# B&R Automation Studio project Soiled_PLC (part 14)

#### pc.st - Implementation code
```iecst
(********************************************************************
 * COPYRIGHT --
 ********************************************************************
 * Program: pr
 * File: pr.st
 * Author: treamsbottom
 * Created: July 16, 2015
 ********************************************************************
 * Implementation of program pr
 ********************************************************************)
//V1.00.1 First Release
PROGRAM _INIT
//Configuration
mySeq						:= 10;		//Sequence number
myIO						:= 191;
myX20IO						:= 6;		// IO for hardwired stops
myPC						:= 1;
myZone						:= 0;
myRelLine					:= 22;
useRequest					:= FALSE; 	//Use the Request bit. Only use when working with x_1_point. otherwise use RequestRelease as the i_bagAtBuffer.
myBuffBag					:= 0; 		//Buffer bag
myBag						:= 255; 	//Buffer Bag
bufferSettleTime			:= 300;

isDecline					:= FALSE; // VC is moving bags down
myOutBag 					:= Line[myRelLine].LastBag;
END_PROGRAM

PROGRAM _CYCLIC
//Inputs
i_carrAtTop					:= X[myIO].X01;
i_carrAtBottom				:= X[myIO].X02;
i_bagArrive					:= X[myIO].X03;
i_bagOnCarriage				:= X[myIO].X04;
i_bagAtBuffer				:= X[myIO].X05;

i_bagAtBufferOut 		:= FALSE; // Any Single bag buffer out IO.
i_bufferOutOpen			:= FALSE;

o_openBuffer			:= FALSE;
o_openCarriageStop		:= FALSE;
moveToIncomingPosition	:= FALSE;
moveToOutgoingPosition	:= FALSE;

Request.PC[myPC]		:= FALSE;
RequestRel.PC[myPC]		:= FALSE;

IF (myBag = 0) THEN
	Alarm[mySeq].Bag	:= mySeq + 10000;
ELSE
	Alarm[mySeq].Bag	:= myBag;
END_IF;

Alarm[mySeq].Name 		:= 0;
Alarm[mySeq].Beacon		:= TRUE;
Alarm[mySeq].Extra		:= 0;
Alarm[mySeq].Time		:= 3000;

//Setup Sequence
step := D[900 + mySeq];
//Setup Pulse contact
pls := (step <> lastStep);
lastStep := step;

//Sequence
IF (step = 0) THEN
	//Disabled
END_IF;

//Step 1 move to bag in position
IF (step = 1) THEN
	moveToIncomingPosition := TRUE;
	IF carrInIncomingPos THEN
		D[900 + mySeq] := 2;
	END_IF
	IF NOT Std.HaltSysZone[myZone] THEN
		Alarm[mySeq].Name := ALM_CARRIAGE_MOVE_FAULT;
	END_IF;
END_IF;

//Wait for at buffer
ton_10ms_SettledBuffer(IN:= i_bagAtBuffer, PT:= bufferSettleTime);
IF (step = 2) THEN
	moveToIncomingPosition := TRUE;
	IF carrInIncomingPos AND NOT Std.HaltSysZone[myZone] AND NOT i_bagOnCarriage AND NOT i_bagArrive THEN
		IF useRequest THEN
			D[900 + mySeq] := 3;
		ELSE
			IF ton_10ms_SettledBuffer.Q THEN
				IF (myBuffBag > 0) THEN
					IF (Bag[myBuffBag].Cat > 0) AND (Bag[myBag].Cat = 0) THEN
						D[900 + mySeq] := 3;
					ELSIF (Bag[myBuffBag].Cat = 0) THEN
						Alarm[mySeq].Name := ALM_BAG_DATA_ERROR;
						Alarm[mySeq].Bag := myBuffBag;
					ELSE
						Alarm[mySeq].Name := ALM_BAG_DATA_ERROR;
					END_IF;
				ELSE
					D[900 + mySeq] := 3;
				END_IF;
			ELSIF (myBuffBag > 0) AND (Bag[myBuffBag].Cat > 0) THEN
				Alarm[mySeq].Name := ALM_BAG_NOT_SETTLED;
			END_IF;
		END_IF;
	ELSIF NOT Std.HaltSysZone[myZone] THEN
		Alarm[mySeq].Name := ALM_SWITCH_FAULT;
	END_IF;
END_IF;

//Open Buffer stop
IF (step = 3) THEN
	moveToIncomingPosition := TRUE;
	IF carrInIncomingPos THEN
		carrInPosLatch := TRUE;
	END_IF;
	releaseValid := (carrInPosLatch AND ((myBag = 0) OR ((Bag[myBag].Cat = 0) AND (Bag[myBuffBag].Cat > 0))));
	o_openBuffer	   := releaseValid AND NOT useRequest;
	Request.PC[myPC]  := releaseValid AND useRequest;
	IF ((i_bagArrive OR i_bagOnCarriage) AND releaseValid) THEN
		IF (myBag > 0) THEN
			Bag[myBag] := Bag[myBuffBag]; //Clear empty buffer bag data if used
			Bag[myBuffBag] := Bag[0];
		END_IF;
		D[900 + mySeq] := 4;
	ELSIF (myBag > 0) THEN
		IF (Bag[myBag].Cat > 0) THEN
			Alarm[mySeq].Name := ALM_BAG_DATA_ERROR;
			Alarm[mySeq].Time := 0;
		ELSIF (Bag[myBuffBag].Cat = 0) THEN
			Alarm[mySeq].Name := ALM_BAG_DATA_ERROR;
			Alarm[mySeq].Bag := myBuffBag;
			Alarm[mySeq].Time := 0;
		ELSE
			Alarm[mySeq].Name  := ALM_BAG_NOT_ARRIVED;
		END_IF;
	ELSIF NOT carrInPosLatch THEN
		Alarm[mySeq].Name  := ALM_SWITCH_FAULT;
	ELSE
		Alarm[mySeq].Name  := ALM_BAG_NOT_ARRIVED;
	END_IF;
END_IF;

// Step 4 Bag settles on carriage..
ton_10ms_SettledCarriage(IN:= i_bagOnCarriage, PT:= 300);
IF (step = 4) THEN
	moveToIncomingPosition := TRUE;
	IF  ton_10ms_SettledCarriage.Q AND NOT Std.HaltSysZone[myZone] AND NOT i_bagArrive THEN
		D[900 + mySeq] := 5;
	ELSIF NOT Std.HaltSysZone[myZone] THEN
		Alarm[mySeq].Name := ALM_BAG_NOT_SETTLED;
	END_IF;
END_IF

// Step 5 move to outgoing position
IF (step = 5) THEN
	moveToOutgoingPosition := TRUE;
	IF carrAtOutgoingPos THEN
		D[900 + mySeq] := 6;
	ELSIF NOT Std.HaltSysZone[myZone] THEN
		Alarm[mySeq].Name := ALM_CARRIAGE_MOVE_FAULT;
	END_IF;
END_IF;

//Step 6 check release condtion.
//Check for line space.
IF (step = 6) THEN
	moveToOutgoingPosition := TRUE;
	releaseValid := (carrAtOutgoingPos AND NOT i_bagAtBufferOut AND NOT i_bufferOutOpen AND ((myBag = 0) OR ((Bag[myBag].Cat > 0) AND (Bag[myOutBag].Cat = 0))));
	IF (myRelLine > 0) THEN
		IF (Line[myRelLine].Clear AND releaseValid) THEN
			C[myRelLine] := 0;
			D[900 + mySeq] := 7;
		END_IF;
		IF NOT carrAtOutgoingPos THEN
			Alarm[mySeq].Name := ALM_CARRIAGE_MOVE_FAULT;
			Alarm[mySeq].Time := 0;
		ELSIF (Line[myRelLine].Clear AND i_bagAtBufferOut) THEN
			Alarm[mySeq].Name := ALM_SWITCH_FAULT;
		ELSIF (myBag > 0) AND (Bag[myBag].Cat = 0) THEN
			Alarm[mySeq].Name := ALM_BAG_DATA_ERROR;
			Alarm[mySeq].Time := 0;
		ELSIF Line[myRelLine].Clear AND (myOutBag > 0) AND (Bag[myOutBag].Cat > 0) THEN
			Alarm[mySeq].Name := ALM_BAG_DATA_ERROR;
			Alarm[mySeq].Bag := myOutBag;
			Alarm[mySeq].Time := 0;
		END_IF;
	ELSE
		RequestRel.PC[myPC] := releaseValid;
		IF EnableRel.PC[myPC] AND releaseValid THEN
			D[900 + mySeq] := 7;
		ELSIF NOT carrAtOutgoingPos THEN
			Alarm[mySeq].Name := ALM_CARRIAGE_MOVE_FAULT;
			Alarm[mySeq].Time := 0;
		ELSIF (myBag > 0) AND (Bag[myBag].Cat = 0) THEN
			Alarm[mySeq].Name := ALM_BAG_DATA_ERROR;
			Alarm[mySeq].Time := 0;
		ELSIF (myOutBag > 0) AND (Bag[myOutBag].Cat > 0) THEN
			Alarm[mySeq].Name := ALM_BAG_DATA_ERROR;
			Alarm[mySeq].Bag := myOutBag;
			Alarm[mySeq].Time := 0;
		END_IF;
	END_IF;
END_IF;

//Step 7 Release bag.
IF (step = 7) THEN
	releaseValid := (NOT i_bagAtBufferOut AND NOT i_bufferOutOpen AND ((myBag = 0) OR ((Bag[myBag].Cat > 0) AND (Bag[myOutBag].Cat = 0))));
	o_openCarriageStop := releaseValid AND NOT Std.HaltSysZone[myZone];
	IF releaseValid THEN
		IF (myBag = 0) THEN
			IF (myRelLine > 0) THEN
				IF Line[myRelLine].Trip THEN
					D[900 + mySeq] := 1;
				END_IF;
			ELSE
				IF NOT EnableRel.PC[myPC] THEN
					D[900 + mySeq] := 1;
				END_IF;
			END_IF;
			IF NOT Std.HaltSysZone[myZone] THEN
				Alarm[mySeq].Name := ALM_BAG_NOT_RELEASED;
			END_IF;
		ELSE//Use tracking
			IF (myRelLine > 0) THEN
				IF Line[myRelLine].Trip THEN
					Bag[myOutBag] := Bag[myBag];
					Bag[myBag] := Bag[0];
					D[900 + mySeq] := 1;
				END_IF;
			ELSE
				IF NOT EnableRel.PC[myPC] AND (Bag[myBag].Cat = 0) THEN // Make sure data is copied out by enabling sequence.
					D[900 + mySeq] := 1;
				ELSIF NOT EnableRel.PC[myPC] AND (Bag[myBag].Cat > 0) THEN
					Alarm[mySeq].Name := ALM_BAG_DATA_ERROR;
				END_IF;
			END_IF;
		END_IF;
	ELSIF NOT carrAtOutgoingPos THEN
		Alarm[mySeq].Name := ALM_CARRIAGE_MOVE_FAULT;
		Alarm[mySeq].Time := 0;
	ELSIF i_bagAtBufferOut AND NOT i_bufferOutOpen THEN
		Alarm[mySeq].Name := ALM_SWITCH_FAULT;
		Alarm[mySeq].Time := 0;
	ELSIF (myBag > 0) THEN
		IF (Bag[myBag].Cat = 0) THEN
			Alarm[mySeq].Name := ALM_BAG_DATA_ERROR;
			Alarm[mySeq].Time := 0;
		ELSIF (Bag[myOutBag].Cat > 0) THEN
			Alarm[mySeq].Name := ALM_BAG_DATA_ERROR;
			Alarm[mySeq].Bag := myOutBag;
			Alarm[mySeq].Time := 0;
		END_IF;
	END_IF;
END_IF;

//Control Position
IF isDecline THEN
	o_moveUp := moveToIncomingPosition;
	o_moveDown := moveToOutgoingPosition;
	carrInIncomingPos := i_carrAtTop;
	carrAtOutgoingPos := i_carrAtBottom;
ELSE
	o_moveDown := moveToIncomingPosition;
	o_moveUp := moveToOutgoingPosition;
	carrInIncomingPos := i_carrAtBottom;
	carrAtOutgoingPos := i_carrAtTop;
END_IF;

//-----------------------------------
//PLC Outputs - adjust TO suit system
//-----------------------------------

Y[myIO].Y06			:= o_openBuffer;
Y[myIO].Y07			:= ((step >= 3) AND (step <= 4) AND carrInIncomingPos); //Safe stop

Y[myX20IO].Y01 		:= (o_moveUp AND NOT i_carrAtTop); //Move carriage up
Y[myX20IO].Y02 		:= (o_moveDown  AND NOT i_carrAtBottom);//Move carriage down
Y[myX20IO].Y03 		:= (o_openCarriageStop AND carrAtOutgoingPos);// Carriage Stop

//Don't allow forcing of carriage movement and carriage stop
YForceDisable[myX20IO].Y01 	:= TRUE;
YForceDisable[myX20IO].Y02 	:= TRUE;
YForceDisable[myX20IO].Y03 	:= TRUE;

//Alarms
timerAlarm(IN := NOT pls AND (Alarm[mySeq].Name > 0),PT:= Alarm[mySeq].Time);

Alarm[mySeq].On 	:= timerAlarm.Q;
Alarm[mySeq].ET 	:= timerAlarm.ET;

END_PROGRAM
```

### Program Logical/BaseStandards/Pneumatic/pic (IEC, version 1.00.3) - *Pneumatic Incline

#### pic.st - Implementation code
```iecst
(********************************************************************
 * COPYRIGHT --
 ********************************************************************
 * Program: pic
 * File: pic.st
 * Author: treamsbottom
 * Created: July 16, 2015
 ********************************************************************
 * Implementation of program pic - Pneumatic Incline
 ********************************************************************)
//V1.00.1 First Release
PROGRAM _INIT
//Configuration
mySeq						:= 22;	//Sequence number
myIO						:= 201;
myZone						:= 0;
myRelLine					:= 22;
myBuffBag					:= 0;
myBag						:= 0;
bufferSettleTime			:= 300;
myPI						:= 1;

myOutBag 					:= Line[myRelLine].LastBag;
END_PROGRAM

PROGRAM _CYCLIC
//Inputs

i_bagInIncline			:= X[myIO].X01;
i_cylinderAtBottom		:= X[myIO].X02;
i_cylinderAtTop			:= X[myIO].X03;
i_bagAtBuffer			:= X[myIO].X04;

i_bagAtBufferOut 		:= FALSE; // Any Single bag buffer out IO.
i_bufferOutOpen			:= FALSE;

o_openBuffer			:= FALSE;
o_cylinderDown			:= FALSE;

Request.PI[myPI]		:= FALSE;
RequestRel.PI[myPI]		:= FALSE;

IF (myBag = 0) THEN
	Alarm[mySeq].Bag	:= mySeq + 10000;
ELSE
	Alarm[mySeq].Bag	:= myBag;
END_IF;

Alarm[mySeq].Name 		:= 0;
Alarm[mySeq].Beacon	:= TRUE;
Alarm[mySeq].Extra		:= 0;
Alarm[mySeq].Time		:= 3000;

//Setup Sequence
step := D[900 + mySeq];
//Setup Pulse contact
pls := (step <> lastStep);
lastStep := step;

//Sequence
IF (step = 0) THEN
	//Disabled
END_IF;

//Wait for at buffer
ton_10ms_SettledBuffer(IN:= i_bagAtBuffer, PT:= bufferSettleTime);
IF (step = 1) THEN
	IF NOT Std.HaltSysZone[myZone] AND i_cylinderAtTop AND NOT i_bagInIncline THEN
		IF useRequest THEN
			D[900 + mySeq] := 2;
		ELSE
			IF ton_10ms_SettledBuffer.Q THEN
				IF (myBuffBag > 0) THEN
					IF (Bag[myBuffBag].Cat > 0) AND (Bag[myBag].Cat = 0) THEN
						D[900 + mySeq] := 2;
					ELSIF (Bag[myBuffBag].Cat = 0) THEN
						Alarm[mySeq].Name := ALM_BAG_DATA_ERROR;
						Alarm[mySeq].Bag := myBuffBag;
					ELSE
						Alarm[mySeq].Name := ALM_BAG_DATA_ERROR;
					END_IF;
				ELSE
					D[900 + mySeq] := 2;
				END_IF;
			ELSIF (myBuffBag > 0) AND (Bag[myBuffBag].Cat > 0) THEN
				Alarm[mySeq].Name := ALM_BAG_NOT_SETTLED;
			END_IF;
		END_IF;
	ELSIF NOT Std.HaltSysZone[myZone] THEN
		Alarm[mySeq].Name := ALM_SWITCH_FAULT;
	END_IF;
END_IF;

//Open Buffer stop
IF (step = 2) THEN
	releaseValid := ((myBag = 0) OR ((Bag[myBag].Cat = 0) AND (Bag[myBuffBag].Cat > 0)));
	o_openBuffer	   := releaseValid AND NOT useRequest;
	Request.PI[myPI]  := releaseValid AND useRequest;
	IF (i_bagInIncline AND releaseValid) THEN
		IF (myBag > 0) THEN
			Bag[myBag] := Bag[myBuffBag]; //Clear empty buffer bag data if used
			Bag[myBuffBag] := Bag[0];
		END_IF;
		D[900 + mySeq] := 3;
	ELSIF (myBag > 0) THEN
		IF (Bag[myBag].Cat > 0) THEN
			Alarm[mySeq].Name := ALM_BAG_DATA_ERROR;
			Alarm[mySeq].Time := 0;
		ELSIF (Bag[myBuffBag].Cat = 0) THEN
			Alarm[mySeq].Name := ALM_BAG_DATA_ERROR;
			Alarm[mySeq].Bag := myBuffBag;
			Alarm[mySeq].Time := 0;
		ELSE
			Alarm[mySeq].Name  := ALM_BAG_NOT_ARRIVED;
		END_IF;
		Alarm[mySeq].Name  := ALM_BAG_NOT_ARRIVED;
	END_IF;
END_IF;

//Let bag settle at base OF incline
ton_10ms_SettledInIncline(IN:= i_bagInIncline, PT:= 300);
IF (step = 3) THEN
	o_openBuffer := NOT useRequest;
	IF  ton_10ms_SettledInIncline.Q AND NOT Std.HaltSysZone[myZone] THEN
		D[900 + mySeq] := 4;
	ELSIF NOT Std.HaltSysZone[myZone] THEN
		Alarm[mySeq].Name := ALM_BAG_NOT_SETTLED;
	END_IF;
END_IF

//Move incline down to collect first trolley
ton_10ms_CylinderDown(IN := i_cylinderAtBottom, PT:=300);
IF (step = 4) THEN
	o_openBuffer := NOT useRequest;
	o_cylinderDown := TRUE;
	IF ton_10ms_CylinderDown.Q THEN
		D[900 + mySeq] := 5;
	END_IF;
	Alarm[mySeq].Name := ALM_SWITCH_FAULT;
END_IF;

//Let cylinder move back to the top.
IF (step = 5) THEN
	o_openBuffer := NOT useRequest;
	IF i_cylinderAtTop THEN
		D[900 + mySeq] := 6;
	END_IF;
	Alarm[mySeq].Name := ALM_SWITCH_FAULT;
END_IF;

//Check for valid release..
//Check for line space.
IF (step = 6) THEN
	releaseValid := (ton_10ms_SettledInIncline.Q AND NOT i_cylinderAtBottom AND NOT i_bagAtBufferOut AND NOT i_bufferOutOpen AND ((myBag = 0) OR ((Bag[myBag].Cat > 0) AND (Bag[myOutBag].Cat = 0))));
	IF (myRelLine > 0) THEN
		IF (Line[myRelLine].Clear AND releaseValid) THEN
			C[myRelLine] := 0;
			D[900 + mySeq] := 7;
		END_IF;
		IF i_cylinderAtBottom OR NOT i_bagInIncline THEN
			Alarm[mySeq].Name := ALM_SWITCH_FAULT;
			Alarm[mySeq].Time := 0;
		ELSIF (Line[myRelLine].Clear AND i_bagAtBufferOut) THEN
			Alarm[mySeq].Name := ALM_SWITCH_FAULT;
		ELSIF (myBag > 0) AND (Bag[myBag].Cat = 0) THEN
			Alarm[mySeq].Name := ALM_BAG_DATA_ERROR;
			Alarm[mySeq].Time := 0;
		ELSIF Line[myRelLine].Clear AND (myOutBag > 0) AND (Bag[myOutBag].Cat > 0) THEN
			Alarm[mySeq].Name := ALM_BAG_DATA_ERROR;
			Alarm[mySeq].Bag := myOutBag;
			Alarm[mySeq].Time := 0;
		END_IF;
	ELSE
		RequestRel.PI[myPI] := releaseValid;
		IF EnableRel.PI[myPI] AND releaseValid THEN
			D[900 + mySeq] := 7;
		ELSIF NOT i_cylinderAtBottom OR NOT i_bagInIncline THEN
			Alarm[mySeq].Name := ALM_SWITCH_FAULT;
			Alarm[mySeq].Time := 0;
		ELSIF (myBag > 0) AND (Bag[myBag].Cat = 0) THEN
			Alarm[mySeq].Name := ALM_BAG_DATA_ERROR;
			Alarm[mySeq].Time := 0;
		ELSIF (myOutBag > 0) AND (Bag[myOutBag].Cat > 0) THEN
			Alarm[mySeq].Name := ALM_BAG_DATA_ERROR;
			Alarm[mySeq].Bag := myOutBag;
			Alarm[mySeq].Time := 0;
		END_IF;
	END_IF;
END_IF;

//Move cylinder down to get 2nd trolley.
IF (step = 7) THEN
	o_cylinderDown := TRUE;
	IF  ton_10ms_CylinderDown.Q THEN
		D[900 + mySeq] := 8;
	END_IF;
	Alarm[mySeq].Name := ALM_SWITCH_FAULT;
END_IF;

//Release bag
IF (step = 8) THEN
	releaseValid := (NOT i_bagAtBufferOut AND NOT i_bufferOutOpen AND ((myBag = 0) OR ((Bag[myBag].Cat > 0) AND (Bag[myOutBag].Cat = 0))));
	o_cylinderDown := NOT releaseValid; // Hold cylinder down if release is not valid.
	IF releaseValid THEN
		IF (myBag = 0) THEN// Not tracking.
			IF (myRelLine > 0) THEN
				IF Line[myRelLine].Trip THEN
					D[900 + mySeq] := 1;
				END_IF;
			ELSE
				IF NOT EnableRel.PI[myPI] THEN
					D[900 + mySeq] := 1;
				END_IF;
			END_IF;
			IF NOT Std.HaltSysZone[myZone] THEN
				Alarm[mySeq].Name := ALM_BAG_NOT_RELEASED;
			END_IF;
		ELSE//Use tracking
			IF (myRelLine > 0) THEN
				IF Line[myRelLine].Trip THEN
					Bag[myOutBag] := Bag[myBag];
					Bag[myBag] := Bag[0];
					D[900 + mySeq] := 1;
				END_IF;
			ELSE
				IF NOT EnableRel.PI[myPI] AND (Bag[myBag].Cat = 0) THEN // Make sure data is copied out by enabling sequence.
					D[900 + mySeq] := 1;
				ELSIF NOT EnableRel.PI[myPI] AND (Bag[myBag].Cat > 0) THEN
					Alarm[mySeq].Name := ALM_BAG_DATA_ERROR;
				END_IF;
			END_IF;
		END_IF;
	ELSIF i_bagAtBufferOut AND NOT i_bufferOutOpen THEN
		Alarm[mySeq].Name := ALM_SWITCH_FAULT;
		Alarm[mySeq].Time := 0;
	ELSIF (myBag > 0) THEN
		IF (Bag[myBag].Cat = 0) THEN
			Alarm[mySeq].Name := ALM_BAG_DATA_ERROR;
			Alarm[mySeq].Time := 0;
		ELSIF (Bag[myOutBag].Cat > 0) THEN
			Alarm[mySeq].Name := ALM_BAG_DATA_ERROR;
			Alarm[mySeq].Bag := myOutBag;
			Alarm[mySeq].Time := 0;
		END_IF;
	END_IF;
END_IF

//-----------------------------------
//PLC Outputs - adjust TO suit system
//-----------------------------------

Y[myIO].Y05 := o_cylinderDown;
Y[myIO].Y06 := o_openBuffer;

//Alarms
timerAlarm(IN := NOT pls AND (Alarm[mySeq].Name > 0),PT:= Alarm[mySeq].Time);

Alarm[mySeq].On 	:= timerAlarm.Q;
Alarm[mySeq].ET 	:= timerAlarm.ET;

END_PROGRAM
```

### Package Logical/BaseStandards/Misc - Misc - Speed Reducer,Pressure relief

### Program Logical/BaseStandards/Misc/ssr (IEC, version 1.00.1) - speed reducer

- Standard Sequence Speed Reducer V1.00.1 ENG.docx (binary file, 203679 bytes)
#### ssr.st - Implementation code
```iecst
(********************************************************************
 * COPYRIGHT --
 ********************************************************************
 * Program: ssr
 * File: ssr.st
 * Author: treamsbottom
 * Created: July 16, 2015
 ********************************************************************
 * Implementation of program ssr
 ********************************************************************)
//V1.00.1 FIRST VERSION
PROGRAM _INIT

END_PROGRAM

PROGRAM _CYCLIC

myHaltSys				:= Std.HaltSysZone[0];

//Inputs
i_bagApproach[1]		:= X[212].X01;

FOR n := 1 TO LOCAL_MAX_SPEED_REDUCERS DO

	ctu_tripCount[n](CU	:= i_bagApproach[n],PV := 2,RESET := ton_10ms_openBrush[n].Q);
	ton_10ms_openBrush[n](IN := NOT myHaltSys AND o_closeBrush[n],PT	:= 300);

	IF (ctu_tripCount[n].CV >= 2) THEN
		o_closeBrush[n] := TRUE;
	END_IF;

	IF ton_10ms_openBrush[n].Q THEN
		o_closeBrush[n] := FALSE;
	END_IF;
END_FOR;

//Outputs
Y[212].Y05		:= o_closeBrush[1];

END_PROGRAM
```

#### ssr.var - Local variables
```iecst
(********************************************************************
 * COPYRIGHT --
 ********************************************************************
 * Program: ssr
 * File: ssr.var
 * Author: treamsbottom
 * Created: July 16, 2015
 ********************************************************************
 * Local variables of program ssr
 ********************************************************************)
VAR
	myHaltSys : BOOL;
	i_bagApproach : ARRAY[0..LOCAL_MAX_SPEED_REDUCERS] OF BOOL;
	n : UINT;
	ctu_tripCount : ARRAY[0..LOCAL_MAX_SPEED_REDUCERS] OF CTU;
	ton_10ms_openBrush : ARRAY[0..LOCAL_MAX_SPEED_REDUCERS] OF TON_10ms;
	o_closeBrush : ARRAY[0..LOCAL_MAX_SPEED_REDUCERS] OF BOOL;
END_VAR
VAR CONSTANT
	LOCAL_MAX_SPEED_REDUCERS : UINT := 1;
END_VAR
```

### Package Logical/BaseStandards/Sorting - *All sorting equipment

### Program Logical/BaseStandards/Sorting/zzCustomerChange (IEC)

#### zzCustomerChange.ab - Implementation code
```automation-basic
(********************************************************************
 * COPYRIGHT -- HP
 ********************************************************************
 * Program: zzCustomerChange
 * File: zzCustomerChange.ab
 * Author: treamsbottom
 * Created: November 18, 2014
 ********************************************************************
 * Implementation of program zzCustomerChange
 ********************************************************************)

PROGRAM _INIT

END_PROGRAM

 PROGRAM _CYCLIC
; Multiple Bank Customer change,UINT
; Use D32[80 + Bank] to send new customer
; Use D32[90 + Bank] for reply

myZone 			= 0
mySeq			= 83
;I_PxStart_Belt[3] = X[3].X04;belt blocked
I_PxEnd_Belt[3] = NOT X[350].X01
I_PxEnd_Belt[4] = NOT X[351].X01
I_PxEnd_Belt[5] = NOT X[351].X02
I_PxEnd_Belt[7] = NOT X[350].X03
I_PxEnd_Belt[8] = NOT X[351].X03
I_PxEnd_Belt[9] = NOT X[351].X04
I_PxEnd_Belt[11] = NOT X[350].X04
I_PxEnd_Belt[12] = NOT X[350].X02

I_InvStatus[2]	= X[360].X06 OR DebugMode
I_InvStatus[3]	= X[360].X07 OR DebugMode
I_InvStatus[4]	= X[360].X08 OR DebugMode
I_InvStatus[5]	= X[361].X01 OR DebugMode
I_InvStatus[7]	= X[361].X02 OR DebugMode
I_InvStatus[8]	= X[361].X03 OR DebugMode
I_InvStatus[9]	= X[361].X04 OR DebugMode
I_InvStatus[11]	= X[361].X05 OR DebugMode
I_InvStatus[12]	= X[361].X06 OR DebugMode

I_MultipleCustomers = (D[900 +  mySeq] = 1)

I_AcceptNewCustomer[1] = X[3].X07
I_AcceptNewCustomer[2] = X[3].X08

myCustBag[1] = 471
myNewCustBag[1] = 472
myCustBag[2] = 473
myNewCustBag[2] = 474

Alarm[mySeq].Name 				= 0
Alarm[mySeq].Bag				= 10083
Alarm[mySeq].Beacon				= TRUE
Alarm[mySeq].Extra				= 0
Alarm[mySeq].Time			  	= 500

LOOP n = 1 TO MAX_BANKS DO
	Bag[myCustBag[n]].Prg = 1
	Bag[myCustBag[n]].Cat = 1 ; Force Cat to stop bag being deleted
	Bag[myCustBag[n]].Bid = n
	Bag[myNewCustBag[n]].Prg = 1
	Bag[myNewCustBag[n]].Cat = 1
	Bag[myNewCustBag[n]].Bid = n+10
	O_CustChange_Lamp[n] = FALSE
	O_CustChange_Piezo[n] = FALSE
	RunBelts[n]	= FALSE
ENDLOOP

LOOP n = 1 TO MAX_BELTS DO
	O_RunBelt[n] = FALSE
	O_SlowBelt[n] = FALSE
ENDLOOP

O_Extend[1] = FALSE
O_Extend[2] = FALSE

O_Retract[1] = FALSE
O_Retract[2] = FALSE

SortingEnable = (D[3] > 0) AND NOT Std.HaltSysZone[myZone]

	;Local Vars for each bank End of first set of sorting belts..
I_End_1st_Belt[1] 		= I_PxEnd_Belt[3]
I_End_1st_Belt[2] 		= I_PxEnd_Belt[7]
;LOOP t = 1 TO 6 DO
;	TON_BeltBlocked[t].IN = I_PxStart_Belt[t]
;	TON_BeltBlocked[t].PT = 150
;	TON_BeltBlocked[t] FUB TON_10ms()
;ENDLOOP
;LOOP t = 1 TO MAX_BANKS DO; IF both px are made and belt is running for more than 6 secs then pulse belt
;
;	TON_RestartBelts[t].IN = (O_RunBelt[t * 3] AND NOT TON_BeltBlocked[t * 3].Q)
;	TON_RestartBelts[t].PT = 300
;	TON_RestartBelts[t] FUB TON_10ms()
;
;	TON_PulseBelt[t].IN = (O_RunBelt[t * 3] AND I_End_1st_Belt[t] AND TON_BeltBlocked[t * 3].Q)
;	TON_PulseBelt[t].PT = 600
;	TON_PulseBelt[t] FUB TON_10ms()
;ENDLOOP
;TON_10ms(NOT PulseOff,500,PulseOn,PulseOnET)
;TON_10ms(PulseOn,200,PulseOff,PulseOffET)

;
;myNextBeltRunning[1]	= ((SortingEnable AND NOT I_End_1st_Belt[1]) OR TON_RestartBelts[1].Q OR (TON_PulseBelt[1].Q AND PulseOn))
;myNextBeltRunning[2]	= ((SortingEnable AND NOT I_End_1st_Belt[2]) OR TON_RestartBelts[2].Q OR (TON_PulseBelt[2].Q AND PulseOn))
;

IF NOT I_MultipleCustomers THEN
	Bag[myNewCustBag[2]].Cus =  Bag[myNewCustBag[1]].Cus
	;CustomerChangeDisplay[2].InputLock = 1	 ;**Is overwritten at end of cyclic code.
ENDIF

LOOP n = 1 TO MAX_BANKS DO
	;Default Display Values
	strcpy(ADR(CustomerChangeDisplay[n].Message),ADR(""))
	CustomerChangeDisplay[n].MessageText_Colour = BgLtGrey + FgBlack
	CustomerChangeDisplay[n].InputLock = 0
	CustomerChangeDisplay[n].InputText_Colour = BgWhite + FgBlack
	CustomerChangeDisplay[n].New_CustomerNo = Bag[myNewCustBag[n]].Cus

	TON_PiezoDelay[n].IN = (CustomerChange[n] = 1)
	TON_PiezoDelay[n].PT = 300
	TON_PiezoDelay[n] FUB TON_10ms()

	IF ((Bag[myNewCustBag[n]].Cus = 0) OR (Bag[myCustBag[n]].Cus = Bag[myNewCustBag[n]].Cus)) THEN
 		CustomerChange[n] = 0
	ENDIF

	CASE CustomerChange[n] OF
		ACTION 0: ; Normal Run Belts as normal
;			strcpy(ADR(CustomerChangeDisplay[n].Message),ADR(""))
;			CustomerChangeDisplay[n].MessageText_Colour = BgLtGrey + FgBlack
;			CustomerChangeDisplay[n].InputLock = 0
;			CustomerChangeDisplay[n].InputText_Colour = BgWhite + FgBlack
			D32[80 + n] = 0
			D32[90 + n] = 0
			RunBelts[n] = SortingEnable
        	IF ((Bag[myCustBag[n]].Cus <> Bag[myNewCustBag[n]].Cus) AND (Bag[myNewCustBag[n]].Cus > 0)) THEN
				CustomerChange[n] = 1
			ENDIF
		ENDACTION

		ACTION 1: ; Stop belt at photocell	and wait for customer change accept.
;			strcpy(ADR(CustomerChangeDisplay[n].Message),ADR("Wait for accept pushbutton"))
;			CustomerChangeDisplay[n].MessageText_Colour = BgLtGrey + FgBlack
;			CustomerChangeDisplay[n].InputLock = 2

			RunBelts[n] = SortingEnable	AND NOT I_End_1st_Belt[n]
			O_CustChange_Lamp[n] = Std.Clock1s
			O_CustChange_Piezo[n] = NOT TON_PiezoDelay[n].Q
			IF I_AcceptNewCustomer[n] THEN
				CustomerChange[n] = 2
			ENDIF
		ENDACTION

		ACTION 2: ;Send new customer request to trackview
			RunBelts[n] = SortingEnable//myNextBeltRunning[n]
			//CustomerChangeDisplay[n].InputLock = 2
			D32[80 + n] = Bag[myNewCustBag[n]].Cus ; Send new customer to trackview

			AutoChangeState = D32[90 + n]
			CASE AutoChangeState OF
				ACTION 0: ;Busy
					//CustomerChangeDisplay[n].MessageText_Colour = BgLtGrey + FgBlack
					//strcpy(ADR(CustomerChangeDisplay[n].Message),ADR("Loading Program - Please Wait"))
					O_CustChange_Lamp[n] = TRUE
					myCustChangeMessageStatus[n] = 99
				ENDACTION

				ACTION 1: ; Ok
					//CustomerChangeDisplay[n].MessageText_Colour = BgLtGrey + FgBlack
					//strcpy(ADR(CustomerChangeDisplay[n].Message),ADR("Program Loaded"))
					Bag[myCustBag[n]].Cus = Bag[myNewCustBag[n]].Cus
					CustomerChange[n] = 0
				ENDACTION

				ACTION 2..3: ; 2 = no program, 3 = invalid
;					IF (AutoChangeState = 2) THEN
;						strcpy(ADR(CustomerChangeDisplay[n].Message),ADR("No Program! Press accept pushbutton"))
;					ELSE
;						strcpy(ADR(CustomerChangeDisplay[n].Message),ADR("Invalid Program! Press accept pushbutton"))
;					ENDIF
;					CustomerChangeDisplay[n].MessageText_Colour = BgLtGrey + FgRed
					O_CustChange_Lamp[n] = Std.Clock500ms
//					myCustChangeMessageStatus[n] = UINT(AutoChangeState)
					IF I_AcceptNewCustomer[n] THEN
						Bag[myCustBag[n]].Cus = Bag[myNewCustBag[n]].Cus
						CustomerChange[n] = 0
					ENDIF
				ENDACTION

				ELSEACTION: ; ERROR!!
				//	strcpy(ADR(CustomerChangeDisplay[n].Message),ADR("ERROR! Press accept pushbutton"))
				//	CustomerChangeDisplay[n].MessageText_Colour = BgLtGrey + FgRed
					O_CustChange_Lamp[n] = Std.Clock500ms
				//	myCustChangeMessageStatus[n] = 4
					IF I_AcceptNewCustomer[n] THEN
						Bag[myCustBag[n]].Cus = Bag[myNewCustBag[n]].Cus
						CustomerChange[n] = 0
					ENDIF
				ENDACTION
			ENDCASE
		ENDACTION

	ENDCASE
ENDLOOP

//**************Belt controls...
	CASE D[983] OF
		ACTION 0://Carousel mode.
			O_Extend[1] = TRUE
			O_Extend[2] = TRUE
        	LOOP n = 1 TO MAX_BELTS DO
				O_RunBelt[n] = SortingEnable AND I_InvStatus[n]
			ENDLOOP
		ENDACTION
		ACTION 1://Retract Both belts
			O_Retract[1] = TRUE
			O_Retract[2] = TRUE
			O_RunBelt[5] =  (SortingEnable AND I_InvStatus[5] AND NOT Stn[41].SP3 AND NOT Stn[41].CloseFlap AND ((Stn[41].QTime = 0) OR NOT I_PxEnd_Belt[5]))
			O_SlowBelt[5] = Stn[41].SP1 AND I_PxEnd_Belt[5]
			O_RunBelt[4] = SortingEnable AND I_InvStatus[4] AND (O_RunBelt[5] OR NOT I_PxEnd_Belt[4])

			O_RunBelt[12] =  (SortingEnable AND I_InvStatus[12] AND NOT Stn[42].SP3 AND NOT Stn[42].CloseFlap AND ((Stn[42].QTime = 0) OR NOT I_PxEnd_Belt[12]))
			O_SlowBelt[12] = Stn[42].SP1 AND I_PxEnd_Belt[12]
			O_RunBelt[11] = SortingEnable AND I_InvStatus[11] AND (O_RunBelt[12] OR NOT I_PxEnd_Belt[11])
			O_RunBelt[9] = SortingEnable AND I_InvStatus[9] AND (O_RunBelt[11] OR NOT I_PxEnd_Belt[9])
			O_RunBelt[8] = SortingEnable AND I_InvStatus[8] AND (O_RunBelt[9] OR NOT I_PxEnd_Belt[8])
		ENDACTION

		ACTION 2://Retract Only SB12
			O_Extend[1] = TRUE
			O_Retract[2] = TRUE
			O_RunBelt[12] =  (SortingEnable AND I_InvStatus[12] AND NOT Stn[42].SP3 AND NOT Stn[42].CloseFlap AND ((Stn[42].QTime = 0) OR NOT I_PxEnd_Belt[12]))
			O_RunBelt[11] = SortingEnable AND I_InvStatus[11] AND (O_RunBelt[12] OR NOT I_PxEnd_Belt[11])
			O_RunBelt[9] = SortingEnable AND I_InvStatus[9] AND (O_RunBelt[11] OR NOT I_PxEnd_Belt[9])
			O_RunBelt[8] = SortingEnable AND I_InvStatus[8] AND (O_RunBelt[9] OR NOT I_PxEnd_Belt[8])

			O_RunBelt[5] = SortingEnable AND I_InvStatus[5] AND (O_RunBelt[10] OR NOT I_PxEnd_Belt[5])
			O_RunBelt[4] = SortingEnable AND I_InvStatus[4] AND (O_RunBelt[5] OR NOT I_PxEnd_Belt[4])
		ENDACTION

		ACTION 3://Retract Only SB5
			O_Retract[1] = TRUE
			O_Extend[2] = TRUE

			O_RunBelt[5] =  (SortingEnable AND I_InvStatus[5] AND NOT Stn[41].SP3 AND NOT Stn[41].CloseFlap AND ((Stn[41].QTime = 0) OR NOT I_PxEnd_Belt[5]))
			O_RunBelt[4] = SortingEnable AND I_InvStatus[4] AND (O_RunBelt[5] OR NOT I_PxEnd_Belt[4])

			O_RunBelt[12] = SortingEnable AND I_InvStatus[12] AND (O_RunBelt[4] OR NOT I_PxEnd_Belt[12])
			O_RunBelt[11] = SortingEnable AND I_InvStatus[11] AND (O_RunBelt[12] OR NOT I_PxEnd_Belt[11])
			O_RunBelt[9] = SortingEnable AND I_InvStatus[9] AND (O_RunBelt[11] OR NOT I_PxEnd_Belt[9])
			O_RunBelt[8] = SortingEnable AND I_InvStatus[8] AND (O_RunBelt[9] OR NOT I_PxEnd_Belt[8])

		ENDACTION

		ACTION 4: //Load only SS42 Split Mode - Retract belt  and stop other on PX
			O_Extend[1] = TRUE
			O_Retract[2] = TRUE
			O_RunBelt[12] =  (SortingEnable AND I_InvStatus[12] AND NOT Stn[42].SP3 AND NOT Stn[42].CloseFlap AND ((Stn[42].QTime = 0) OR NOT I_PxEnd_Belt[12]))
			O_RunBelt[11] = SortingEnable AND I_InvStatus[11] AND (O_RunBelt[12] OR NOT I_PxEnd_Belt[11])
			O_RunBelt[9] = SortingEnable AND I_InvStatus[9] AND (O_RunBelt[11] OR NOT I_PxEnd_Belt[9])
			O_RunBelt[8] = SortingEnable AND I_InvStatus[8] AND (O_RunBelt[9] OR NOT I_PxEnd_Belt[8])

			O_RunBelt[5] = FALSE
			O_RunBelt[4] = SortingEnable AND I_InvStatus[4] AND  NOT I_PxEnd_Belt[4]
		ENDACTION
		ACTION 5:////Load only SS41 Split Mode - Retract belt  and stop other on PX
			O_Retract[1] = TRUE
			O_Extend[2] = TRUE

			O_RunBelt[5] =  (SortingEnable AND I_InvStatus[5] AND NOT Stn[41].SP3 AND NOT Stn[41].CloseFlap AND ((Stn[41].QTime = 0) OR NOT I_PxEnd_Belt[5]))
			O_RunBelt[4] = SortingEnable AND I_InvStatus[4] AND (O_RunBelt[5] OR NOT I_PxEnd_Belt[4])

			O_RunBelt[12] = FALSE//SortingEnable AND I_InvStatus[12] AND (O_RunBelt[4] OR NOT I_PxEnd_Belt[12])
			O_RunBelt[11] = SortingEnable AND I_InvStatus[11] AND  NOT I_PxEnd_Belt[11]
			O_RunBelt[9] = SortingEnable AND I_InvStatus[9] AND (O_RunBelt[11] OR NOT I_PxEnd_Belt[9])
			O_RunBelt[8] = SortingEnable AND I_InvStatus[8] AND (O_RunBelt[9] OR NOT I_PxEnd_Belt[8])
		ENDACTION
		ACTION 6:////Split mode = NO belts retracted.
			O_Extend[1] = TRUE
			O_Extend[2] = TRUE

			O_RunBelt[5] = FALSE
			O_RunBelt[4] = SortingEnable AND I_InvStatus[4] AND  NOT I_PxEnd_Belt[4]

			O_RunBelt[12] = FALSE//SortingEnable AND I_InvStatus[12] AND (O_RunBelt[4] OR NOT I_PxEnd_Belt[12])
			O_RunBelt[11] = SortingEnable AND I_InvStatus[11] AND  NOT I_PxEnd_Belt[11]
			O_RunBelt[9] = SortingEnable AND I_InvStatus[9] AND (O_RunBelt[11] OR NOT I_PxEnd_Belt[9])
			O_RunBelt[8] = SortingEnable AND I_InvStatus[8] AND (O_RunBelt[9] OR NOT I_PxEnd_Belt[8])
		ENDACTION

	ENDCASE

//First sorting belts before platform...
O_RunBelt[3] := SortingEnable AND I_InvStatus[3] AND RunBelts[1] AND (O_RunBelt[4] OR NOT I_PxEnd_Belt[3])
O_RunBelt[2] := O_RunBelt[3] AND I_InvStatus[2]
O_RunBelt[7] := SortingEnable AND I_InvStatus[7] AND RunBelts[2] AND (O_RunBelt[8] OR NOT I_PxEnd_Belt[7])

I_InvStatus[1] = TRUE
I_InvStatus[6] = TRUE
I_InvStatus[10] = TRUE

LOOP n = 1 TO MAX_BELTS DO
	IF NOT I_InvStatus[n] THEN
		Alarm[mySeq].Name = almMotorOverload
		Alarm[mySeq].Time = 0
	ENDIF
EXITIF 	(Alarm[mySeq].Name > 0)
ENDLOOP

TimerAlarm.IN = (Alarm[mySeq].Name > 0)
TimerAlarm.PT = Alarm[mySeq].Time
TimerAlarm FUB TON_10ms()
Alarm[mySeq].On = TimerAlarm.Q
Alarm[mySeq].ET = TimerAlarm.ET

Y[362].Y02 	= O_RunBelt[2]	//1 ,2
Y[362].Y04	= O_RunBelt[3]  //3
Y[362].Y05	= O_RunBelt[4]  //4
Y[362].Y07	= O_RunBelt[5]  //5
Y[363].Y02	= O_RunBelt[7]  //7
Y[363].Y04	= O_RunBelt[8]  //8
Y[363].Y05	= O_RunBelt[9]  //9
Y[363].Y07	= O_RunBelt[11] //10,11
Y[364].Y01	= O_RunBelt[12] //12

Y[362].Y08 = O_SlowBelt[5]
Y[364].Y02 = O_SlowBelt[12]

Y[3].Y01	= O_CustChange_Lamp[1]
Y[3].Y02	= O_CustChange_Piezo[1]// AND Std.Clock500ms
Y[3].Y03	= O_CustChange_Lamp[2]
Y[3].Y04 	= O_CustChange_Piezo[2]// AND Std.Clock500ms

Y[351].Y07	= O_Retract[1]
Y[351].Y08	= O_Extend[1]
Y[350].Y07	= O_Retract[2]
Y[350].Y08	= O_Extend[2]

END_PROGRAM
```

#### zzCustomerChange.var - Local variables
```iecst
(********************************************************************
 * COPYRIGHT -- HP
 ********************************************************************
 * Program: zzCustomerChange
 * File: zzCustomerChange.var
 * Author: treamsbottom
 * Created: November 18, 2014
 ********************************************************************
 * Local variables of program zzCustomerChange
 ********************************************************************)
VAR CONSTANT
	MAX_BANKS : USINT := 2;
	MAX_BELTS : USINT := 12;
END_VAR
VAR
	I_PxEnd_Belt : ARRAY[0..MAX_BELTS] OF BOOL;
	I_MultipleCustomers : BOOL;
	O_RunBelt : ARRAY[0..MAX_BELTS] OF BOOL;
	I_AcceptNewCustomer : ARRAY[0..MAX_BANKS] OF BOOL;
	n : UINT;
	O_CustChange_Piezo : ARRAY[0..MAX_BANKS] OF BOOL;
	O_CustChange_Lamp : ARRAY[0..MAX_BANKS] OF BOOL;
	myZone : UINT;
	SortingEnable : BOOL;
	I_End_1st_Belt : ARRAY[0..MAX_BANKS] OF BOOL;
	CustomerChange : ARRAY[0..MAX_BANKS] OF UINT;
	RunBelts : ARRAY[0..MAX_BELTS] OF BOOL;
	TON_PiezoDelay : ARRAY[0..MAX_BANKS] OF TON_10ms;
	AutoChangeState : UDINT;
	myCustChangeMessageStatus : ARRAY[0..MAX_BANKS] OF UINT;
	myCustBag : ARRAY[0..MAX_BANKS] OF UINT;
	myNewCustBag : ARRAY[0..MAX_BANKS] OF UINT;
	BgRed : UINT;
	BgOrange : UINT;
	BgGreen : UINT;
	FgBlack : UINT;
	BgLtGrey : UINT;
	FgRed : UINT;
	BgWhite : UINT;
	myNextBeltRunning : ARRAY[0..MAX_BELTS] OF BOOL;
	I_PxStart_Belt : ARRAY[0..MAX_BELTS] OF BOOL;
	TON_BeltBlocked : ARRAY[0..MAX_BELTS] OF TON_10ms;
	t : INT;
	TON_PulseBelt : ARRAY[0..MAX_BELTS] OF TON_10ms;
	TON_RestartBelts : ARRAY[0..MAX_BELTS] OF TON_10ms;
	PulseOff : BOOL;
	PulseOn : BOOL;
	PulseOnET : UDINT;
	PulseOffET : UDINT;
	I_InvStatus : ARRAY[0..MAX_BELTS] OF BOOL;
	O_Extend : ARRAY[0..2] OF BOOL;
	O_Retract : ARRAY[0..2] OF BOOL;
	mySeq : UINT;
	TimerAlarm : TON_10ms;
	O_SlowBelt : ARRAY[0..MAX_BELTS] OF BOOL;
END_VAR
```

### Program Logical/BaseStandards/Sorting/41_stnsa1 (IEC) - *Sorting Stations--

#### stnsa.ab
```automation-basic
PROGRAM _CYCLIC
(* cyclic program *)

;Honeycombe Sorting Station Control
;----------------------------------------------------
;Revision 1.00 10/01/2002 D.J. First Issue
;Revision 2.00 07/02/2005 D.J. Removed Stn Mix
;Revision 3.00 22/08/2006 D.J. Changed to timer array
;----------------------------------------------------

mySeq = 40
Bank = 1

;Timers
OpenTime  = 700
CloseTime = 700

ContinuousSort = TRUE;(D[994] = 0)

;Lamp Test from TrackView
IF (BIT_TST(D[998],0) = 1) THEN
	LampTest = TRUE

ELSE
	LampTest = FALSE
ENDIF

I_PartLoad[1] = X[301].X01
I_PartLoad[2] = X[301].X02
I_PartLoad[3] = X[303].X01
I_PartLoad[4] = X[303].X02
I_PartLoad[5] = X[305].X01
I_PartLoad[6] = X[305].X02
I_PartLoad[7] = X[307].X01
I_PartLoad[8] = X[307].X02
I_PartLoad[9] = X[309].X01
I_PartLoad[10] = X[309].X02
I_PartLoad[11] = X[311].X01
I_PartLoad[12] = X[311].X02
I_PartLoad[13] = X[313].X01
I_PartLoad[14] = X[313].X02
I_PartLoad[15] = X[315].X01
I_PartLoad[16] = X[315].X02
I_PartLoad[17] = X[317].X01
I_PartLoad[18] = X[317].X02
I_PartLoad[19] = X[319].X01
I_PartLoad[20] = X[319].X02

LOOP x = 1 TO Ldg[Bank].NoStations DO
		n = Ldg[Bank].Stations[x]

		;Parts Loads
		TimerPartLoad[n].IN		= I_PartLoad[n]
		TimerPartLoad[n].PT		= 100
		TimerPartLoad[n] FUB TON_10ms()

		IF TimerPartLoad[n].Q THEN
			D[800 + n] = 1
		ENDIF

		;Bag open timers
		TimerOpen[n].IN 		= OpenBag[n]
		TimerOpen[n].PT			= OpenTime
		TimerOpen[n] FUB TON_10ms()

		BagOpened[n] 			= TimerOpen[n].Q
		BagOpenedET[n]			= TimerOpen[n].ET

		;Bag closed timers
		TimerClosed[n].IN 		= NOT OpenBag[n]
		TimerClosed[n].PT		= CloseTime
		TimerClosed[n] FUB TON_10ms()

		BagClosed[n] 			= TimerClosed[n].Q
		BagClosedET[n]			= TimerClosed[n].ET

		;Update bag weight
		StnBag = LDG_GetBagFromStation(Std.StationBagsStart,n)
		Bag[StnBag].Wgt 		= Stn[n].Weight
		Bag[StnBag].Cnt 		= Stn[n].Count

		;Update Bag ID if cleared or zero
		IF ((BidStn > 0) AND (Bag[StnBag].Bid = 0) AND (Bag[StnBag].Cat > 0)) THEN
			Bag[StnBag].Bid = UINT(BidStn)
			BidStn			= 0
		ENDIF

		;Move bags from Display buffer position into Search array,,
		myDisplayBag = LDG_GetBagFromStation(Std.StationBagDisplay,n)

		;Keep Weight Live on Display
		Bag[myDisplayBag].Wgt = Stn[n].Weight
		Update = FALSE
		IF (Bag[StnBag].Cat <> Bag[myDisplayBag].Cat) THEN
			Update = TRUE
		ELSE IF (Bag[StnBag].Cus <> Bag[myDisplayBag].Cus) THEN
			Update = TRUE
		ELSE IF (Bag[StnBag].Prg <> Bag[myDisplayBag].Prg) THEN
			Update = TRUE
		ENDIF
		IF (Bag[myDisplayBag].Cat = Std.MaxCats) THEN
			Update = FALSE ; Do not update bag if Empty Bag is assigned.
			CloseFlap[n] = TRUE
		ELSE
			CloseFlap[n] = FALSE
		ENDIF

		;Flap close after above SP2 for 1 second
		TimerFlapClose[n].IN 	= Stn[n].SP2 AND (Bag[myDisplayBag].Cat <> Std.MaxCats)
		TimerFlapClose[n].PT	= 200 ;4 sec
		TimerFlapClose[n] FUB TON_10ms()

		IF ContinuousSort THEN
			AutoPurgeTrig[n].CLK = Update
			AutoPurgeTrig[n] FUB R_TRIG()
			IF AutoPurgeTrig[n].Q THEN
				newBag[n] = TRUE
			ENDIF

			IF (newBag[n] AND Std.AutoPurge AND NOT Stn[n].CloseFlap AND NOT Stn[n].ManualRelease AND NOT Stn[n].Purge AND NOT Stn[n].PurgeReverse)THEN
				D[800 + n] = 2 ; Bag change detected automatically purge the station... Weight is check in ZZstn
				newBag[n] = FALSE
			ENDIF

			IF ((NOT Stn[n].CloseFlap AND NOT Stn[n].ManualRelease AND NOT Stn[n].Purge AND NOT Stn[n].PurgeReverse AND (D[800 + n] = 0)) OR  (Bag[StnBag].Cat = 0)) THEN ;AND NOT Stn[n].SP2 THEN
				IF Update THEN;(Update AND (n <> 12)) THEN
					myBid = Bag[StnBag].Bid
					Bag[StnBag] = Bag[myDisplayBag]
					Bag[StnBag].Bid = myBid
				ENDIF
			ENDIF
		ELSE
			IF Update THEN
				myBid = Bag[StnBag].Bid
				Bag[StnBag] = Bag[myDisplayBag]
				Bag[StnBag].Bid = myBid
			ENDIF
		ENDIF

		;Ensure Display Bag has a  Bag ID
		IF ((BidStn > 0) AND (Bag[myDisplayBag].Bid = 0) AND  (Bag[myDisplayBag].Cat > 0)) THEN
			Bag[myDisplayBag].Bid = UINT(BidStn)
			BidStn			= 0
		ENDIF

		Alarm[mySeq + n].Name 		= 0
		Alarm[mySeq + n].Bag		= StnBag
		Alarm[mySeq + n].Beacon	= TRUE
		Alarm[mySeq + n].Extra		= 0
		Alarm[mySeq + n].Time		= 4000

		Stn[n].LampOn 		= FALSE
		Stn[n].GreenLamp	= FALSE

		STEP = D[900 + mySeq + n]
		;Setup Pulse contact
		PLS[n] = (STEP <> LASTSTEP[n])
		LASTSTEP[n] = STEP

		;Step 0 - Disabled
		IF (STEP = 0) THEN
			Stn[n].LampOn = TRUE
			Stn[n].CloseFlap = ((Bag[StnBag].Cat <> Bag[myDisplayBag].Cat))
			Stn[n].QTime = 0
			Stn[n].ManualRelease = 0
			Stn[n].Purge = 0
			;Disabled
		ENDIF

		IF (STEP = 1) THEN
			Stn[n].LampOn = TRUE
			Stn[n].GreenLamp = FALSE
			Stn[n].CloseFlap = TRUE
			myStnReg = (n > 32)
			IF (myStnReg = 0)THEN
				myStnBit =	n - 1
			ELSE IF (myStnReg = 1)THEN
				myStnBit = 	n - 33
			ELSE
				myStnBit = 0
			ENDIF
			Std.PurgeBank[Bank].StationsStatus[myStnReg] = BIT_CLR(Std.PurgeBank[Bank].StationsStatus[myStnReg],myStnBit)

	;		Stn[n].Purge = FALSE
	;		Stn[n].PurgeReverse = FALSE
			IF D[900 + Std.StationBankReg + Bank] = n THEN
				D[900 + Std.StationBankReg + Bank] = 0
			ENDIF
			IF BagClosed[n] THEN
				D[900 + mySeq + n] = 2
			ENDIF
			Alarm[mySeq + n].Name = almStationNotClosed
		ENDIF

		IF (STEP = 2) THEN
			Stn[n].LampOn = ((Stn[n].SP1 AND Std.Clock2s) OR Stn[n].SP2 OR (Stn[n].SP3 AND Std.Clock200ms))
			Stn[n].GreenLamp = ((NOT Stn[n].SP2 AND NOT Stn[n].SP3) OR TimerFlapClose[n].Q)
			;Close the flaps when the bag is above SP2
			IF TimerFlapClose[n].Q OR Stn[n].ManualRelease OR Stn[n].Purge OR Stn[n].PurgeReverse THEN
				Stn[n].CloseFlap 	= ContinuousSort
			ENDIF
			;Stop flap closing / re-open is bag below 3kg
			IF (Stn[n].Weight < 30) THEN
				Stn[n].CloseFlap 	= FALSE
			ENDIF
			IF ((D[900 + Std.StationBankReg + Bank] = n) AND Ldg[Bank].EnableStnRelease) THEN
				D[900 + mySeq + n] = 3
			ENDIF
			IF ((Bag[StnBag].Prg > 0) AND Stn[n].SP3) THEN
				Alarm[mySeq + n].Name = almBagOverWeight
			ENDIF
		ENDIF

		IF (STEP = 3) THEN
			Stn[n].LampOn = TRUE
			Stn[n].CloseFlap = ContinuousSort
			Stn[n].GreenLamp = TimerFlapClose[n].Q

			AllowRelease[n]  = TRUE

			IF (BagOpened[n] AND ((Stn[n].Weight < 30) OR Test.Stations) AND Ldg[Bank].BeltHasRun) THEN
				Stn[n].QTime 	= 0
				D[900 + mySeq + n] = 1
			ENDIF
			IF (Stn[n].Weight >= 30) THEN
				Alarm[mySeq + n].Name = almStationNotEmpty
			ENDIF
		ELSE
			AllowRelease[n]= FALSE
		ENDIF

		OpenBag[n] = AllowRelease[n];(STEP = 3)

		;Lamp Test
		IF LampTest THEN
			Stn[n].LampOn = TRUE
		ENDIF

		;Alarm timer
		TimerAlarm[n].IN 	= NOT PLS[n] AND (Alarm[mySeq + n].Name > 0)
		TimerAlarm[n].PT	= Alarm[mySeq + n].Time
		TimerAlarm[n] FUB TON_10ms()

		Alarm[mySeq + n].ET	= TimerAlarm[n].ET
		Alarm[mySeq + n].On 	= TimerAlarm[n].Q

;	Y[300 + n].Y07 = Stn[n].LampOn
;	Y[300 + n].Y05 = Stn[n].CloseFlap OR testClose
;	Y[300 + n].Y06 = Stn[n].GreenLamp
;	Y[300 + n].Y04 = OpenBag[n]

ENDLOOP

;Outputs
;-------
Y[31].Y05 = OpenBag[1]
Y[31].Y06 = OpenBag[2]
Y[31].Y07 = OpenBag[3]
Y[31].Y08 = OpenBag[4]
Y[31].Y13 = OpenBag[5]
Y[31].Y14 = OpenBag[6]
Y[31].Y15 = OpenBag[7]
Y[31].Y16 = OpenBag[8]
Y[32].Y05 = OpenBag[9]
Y[32].Y06 = OpenBag[10]
Y[32].Y07 = OpenBag[11]
Y[32].Y08 = OpenBag[12]
Y[32].Y13 = OpenBag[13]
Y[32].Y14 = OpenBag[14]
Y[32].Y15 = OpenBag[15]
Y[32].Y16 = OpenBag[16]

Y[31].Y01 = Stn[1].LampOn
Y[31].Y02 = Stn[2].LampOn
Y[31].Y03 = Stn[3].LampOn
Y[31].Y04 = Stn[4].LampOn
Y[31].Y09 = Stn[5].LampOn
Y[31].Y10 = Stn[6].LampOn
Y[31].Y11 = Stn[7].LampOn
Y[31].Y12 = Stn[8].LampOn
Y[32].Y01 = Stn[9].LampOn
Y[32].Y02 = Stn[10].LampOn
Y[32].Y03 = Stn[11].LampOn
Y[32].Y04 = Stn[12].LampOn
Y[32].Y09 = Stn[13].LampOn
Y[32].Y10 = Stn[14].LampOn
Y[32].Y11 = Stn[15].LampOn
Y[32].Y12 = Stn[16].LampOn

END_PROGRAM
```

### Program Logical/BaseStandards/Belts/18_stb1 (IEC) - *For Reference only-- Adjust as required.

#### belt.var
```iecst
VAR
	myPrg : USINT;
	BeltAddTimeArray : ARRAY[0..59] OF UINT;
	mySeq : UINT;
	myOtherBeltSeq : UINT;
	myLuBag : UINT;
	myVCBag : UINT;
	PurgeBagIndex : UINT;
	Bank : UINT;
	myBelt : UINT;
END_VAR
VAR RETAIN
	MinBeltRunCV : UINT;
END_VAR
VAR
	STEP : UINT;
	n : UINT;
	myZone : UINT;
	myWgt : UINT;
	StnBag : UINT;
	LASTSTEP : UINT;
	PurgeReverseBagIndex : UINT;
	myOutBag : UINT;
	myOppBeltBag : UINT;
	BeltAddTime : UINT;
	BeltRunTime : UINT;
	VCBag : UINT;
	myBank : UINT;
	myBag : UINT;
	TrackingOkET : UDINT;
	myCus : UDINT;
	LinenDetectedRevET : UDINT;
	myCat : UDINT;
	BeltClearReverseET : UDINT;
	LinenDetectedReverseET : UDINT;
	BeltOKET : UDINT;
	TimerAlarm : TON_10ms;
	LinenIsDetectedET : TIME;
	LargeLoadClearET : TIME;
	Step6ET : TIME;
	LinenDetectedET : TIME;
	BeltClearET : TIME;
	MinimumRunET : TIME;
	myOppositeBelt : INT;
	CountValue : INT;
	WeightValue : INT;
	b : INT;
	MixCust : BOOL;
	BeltOK : BOOL;
	O_Reverse : BOOL;
	Purge : BOOL;
	LinenIsDetected : BOOL;
	MinimumRun : BOOL;
	PhotocellsClear : BOOL;
	MinBeltRunET : BOOL;
	O_SlowBelt : BOOL;
	LinenDetectedReverse : BOOL;
	BeltRunning : BOOL;
	PurgeReverse : BOOL;
	Stb2_Running : BOOL;
	LargeLoadClear : BOOL;
	I_PhotoLarge : BOOL;
	BeltClearReverse : BOOL;
	I_LinenAtEndSTB3 : BOOL;
	RunBelt : BOOL;
	I_PhotoBottom : BOOL;
	O_RunBelt : BOOL;
	LinenDetected : BOOL;
	StationOpen : BOOL;
	I_PhotoTop : BOOL;
	PLS : BOOL;
	MinBeltRun : BOOL;
	WeightValid : BOOL;
	I_DisableLoadingUnit : BOOL;
	LinenDetectedRev : BOOL;
	RunSlow : BOOL;
	I_PhotoReverse : BOOL;
	CountValid : BOOL;
	BeltClear : BOOL;
	TrackingOk : BOOL;
	myOtherBeltRunning : BOOL;
	myStnReg : UINT;
	myStnBit : UINT;
	myTimeStamp : DATE_AND_TIME;
	myHttp : UINT;
	catString : STRING[15];
	cusString : STRING[15];
	wgtString : STRING[15];
	batchString : STRING[32];
	requestURL : STRING[254];
	responseData : ARRAY[0..49] OF USINT;
	commaPos : INT;
	I_InvStatus : BOOL;
	myBagNumber : UINT;
	MixCats : BOOL;
	MixCusts : BOOL;
	MixProgs : BOOL;
	stnNo : USINT;
END_VAR
```

#### beltCyclic.ab
```automation-basic
PROGRAM _INIT
	_setBeltTime

END_PROGRAM

PROGRAM _CYCLIC
 	(* cyclic program *)

;Sequence 2 - Transfer Belt 1 from Stations 1-8

;-----------------------------------------
;Revision 1.00 18/01/2006 D.J. First Issue
;-----------------------------------------

;Inputs and Outputs
;-----------------

myBank 			= 1
myBelt			= 1
mySeq			= 18
myBag			= 220
myOutBag		= 225
myZone			= 1

MixCats			= (D[369] > 0)
MixCusts		= (D[366] > 0)	;Allow mixing of customers?
MixProgs		= (D[367] > 0)	;Allow mixing of Programs?

;I_PhotoBottom		      	= X[3].X08
I_PhotoTop   		      	= X[21].X08
I_PhotoReverse            	= FALSE
I_InvStatus					= X[361].X07

;Belt add times in an array for each station as station number will not work..
;LOOP n = 20 DOWNTO 1 DO
;	BeltAddTimeArray[n]		= n
;ENDLOOP

RequestRel.TransferBelt[myBelt]		  	= FALSE
Request.TransferBelt[myBelt]		    = FALSE

O_RunBelt 					= FALSE
O_Reverse					  = FALSE
O_SlowBelt					= FALSE

;Check all stations are closed.
StationOpen = FALSE
LOOP n = 1 TO Ldg[myBank].NoStations DO
	stnNo = Ldg[myBank].Stations[n]
	IF (D[940 + stnNo] = 3) THEN
		StationOpen = TRUE
	ENDIF
ENDLOOP

Alarm[mySeq].Name 				= 0
Alarm[mySeq].Bag				= myBag
Alarm[mySeq].Beacon				= TRUE
Alarm[mySeq].Extra				= 0
Alarm[mySeq].Time			  	= 5000

n = D[900 + Std.StationBankReg + myBank] ;Selected Station

STEP = D[900 + mySeq]
;Setup Pulse contact
PLS = (STEP <> LASTSTEP)
LASTSTEP = STEP

;Step 0 - Disabled
IF STEP = 0 THEN
	;Disabled
ENDIF

;Step 1 - Check no stations are releasing
IF STEP = 1 THEN
	;Don't allow stations to release
	Ldg[myBank].EnableStnRelease = FALSE
	Std.PurgeBank[myBank].PurgeOn = 0 ; Clear to display Purge
	Std.PurgeBank[myBank].StationsStatus[0] = 0 ;trackview TO display Purge
	Std.PurgeBank[myBank].StationsStatus[1] = 0
	;No Station Releaseng and switched on
	IF (NOT StationOpen AND (D[mySeq] > 0)) THEN
		IF (Bag[myBag].Cat = 0) THEN
			D[900 + mySeq] = 2 ;No Bag on belt
		ELSE
			D[900 + mySeq] = 4 ;Bag on belt
		ENDIF
	ENDIF
	Alarm[mySeq].Name = almNoAlarm
ENDIF

;Step 2 - Enable Station search
IF STEP = 2 THEN
	IF (Bag[myBag].Cat > 0) THEN
		D[900 + mySeq] = 4
	ENDIF
	;Check each station to see if a manual destination has been set
	LOOP n = 1 to Ldg[myBank].NoStations DO

		//StnBag = Std.StationBagsStart + Ldg[myBank].Stations[n] - 1
		StnBag = LDG_GetBagFromStation(Std.StationBagsStart,n)

		IF ((Bag[StnBag].Dst > 0) AND (Bag[StnBag].Dst < 99) AND (D[mySeq] > 0)) THEN ;Dest 99 = Empty Bag in station
			Stn[n].DestManual = Bag[StnBag].Dst
		ELSE
			Stn[n].DestManual = 0
		ENDIF
		;For pairing set number of spaces to search for
		Stn[n].SpacesRequired = 1 ;D[2000 + Bag[StnBag].Prg]

	ENDLOOP

	;Station Search

	IF ((Ldg[myBank].Search = 0) AND (D[mySeq] > 0) AND NOT Std.HaltSysZone[myZone])  THEN
		Ldg[myBank].Search = 1
		PurgeBagIndex = 0
	ELSE IF ((Ldg[myBank].Search = 2) AND (Ldg[myBank].Found > 0)) THEN ;
		IF (Ldg[myBank].Found < 97) THEN
			D[900 + Std.StationBankReg + myBank] 	= Ldg[myBank].Found
			n 	= D[900 + Std.StationBankReg + myBank]
;		ELSE IF (Ldg[myBank].Found = 98) OR (Ldg[myBank].Found = 97) THEN ; Reverse belt
;			D[900 + mySeq] = 9
;			GOTO ExitStep2 ; Ignore the rest of Step 2
		ELSE
;			IF (Ldg[myBank].Found = 98) OR (Ldg[myBank].Found = 97) THEN
;				Ldg[myBank].Line = 21 ; Set Destination to SDC1
;			ENDIF
			Purge = TRUE

			n = LDG_GetStationFromBag(Std.StationBagsStart,Std.PurgeBank[myBank].PurgeBatch[PurgeBagIndex])
			IF (n = 0) OR (n > Ldg[myBank].Stations[Ldg[myBank].NoStations]) THEN
				Ldg[myBank].Search = 0
				GOTO ExitStep2
			ENDIF
			D[900 + Std.StationBankReg + myBank] = n
			Std.PurgeBank[myBank].PurgeOn = 1 ; Send to trackview to display Purge
			myStnReg = (n > 32)
			IF (myStnReg = 0)THEN
				myStnBit =	n - 1
			ELSE IF (myStnReg = 1)THEN
				myStnBit = 	n - 33
				ELSE
				myStnBit = 0
			ENDIF
			Std.PurgeBank[myBank].StationsStatus[myStnReg] = BIT_SET(Std.PurgeBank[myBank].StationsStatus[myStnReg],myStnBit)
			;Get highest belt add time... Use array as station numbers are opposite to distanct
			IF BeltAddTimeArray[n] > BeltAddTime THEN
				BeltAddTime = BeltAddTimeArray[n]
			ENDIF
		ENDIF
		StnBag = LDG_GetBagFromStation(Std.StationBagsStart,n)
		;Clear the release button count if used
		Stn[n].ManualRelease 	= FALSE
		Stn[n].Purge 			= FALSE
		Stn[n].PurgeReverse	 	= FALSE
		Stn[n].PBCount 			= 0
		;------Write Report------
	;	IF Std.StationReports AND (Ldg[myBank].Found <> 98) AND (Ldg[myBank].Found <> 97)THEN
        IF Std.StationReports THEN
			IF (ReportLoading[n].Cat = 0)  THEN
				IF Purge THEN
					IF (PurgeBagIndex < Std.PurgeBank[myBank].PurgeBagQty) THEN
						PurgeBagIndex = PurgeBagIndex + 1
					ENDIF
				ENDIF
				WeightValue = Stn[n].Weight - INT(StnPrev[n].Wgt)
				WeightValid = (WeightValue > 0)

				;Check if anything has been added and current weight is not less than the previous
				CountValue = Stn[n].Count - INT(StnPrev[n].Cnt)
				CountValid = (CountValue > 0)
				IF (WeightValid OR CountValid) THEN
					;Ensure valid values as we report on either a weight or count change
					IF (WeightValue < 0) THEN
						WeightValue = 0
					ENDIF

					IF (CountValue < 0) THEN
						CountValue = 0
					ENDIF
					myTimeStamp = CurrentTimestamp
;					ReportLoading[n].Prg = Bag[StnBag].Prg 			;Program
;					ReportLoading[n].Cat = Bag[StnBag].Cat			;Category
;					ReportLoading[n].Cus = Bag[StnBag].Cus			;Customer
;					ReportLoading[n].Wgt = UINT(WeightValue)		;Weight
;					ReportLoading[n].Cnt = UINT(CountValue)			;Count
;					ReportLoading[n].Stn = n         				;Station
;					ReportLoading[n].Mcn = 0						;Machine
;					ReportLoading[n].Bid = Bag[StnBag].Bid			;Batch ID
;					ReportLoading[n].TimeStamp = myTimeStamp

				ENDIF
			ENDIF
		ELSE
			myTimeStamp = CurrentTimestamp
			IF Purge THEN
				IF (PurgeBagIndex < Std.PurgeBank[myBank].PurgeBagQty) THEN
					PurgeBagIndex = PurgeBagIndex + 1
				ENDIF
			ENDIF
		ENDIF

		;Set Previous Cat and Cus to Current and Clear Weight and Count
		StnPrev[n].Prg 	= Bag[StnBag].Prg
		StnPrev[n].Cat 	= Bag[StnBag].Cat
		StnPrev[n].Cus 	= Bag[StnBag].Cus
		StnPrev[n].Wgt 	= 0
		StnPrev[n].Cnt 	= 0
		StnPrev[n].Bid 	= Bag[StnBag].Bid

		Ldg[myBank].EnableStnRelease = TRUE
		;Clear Manual Release and Count
		Stn[n].ManualRelease 	= FALSE
		Stn[n].Count			= 0
		BeltAddTime = BeltAddTimeArray[n]
		;Keep A record of purged bags to attach the data for the biggest loads
		IF Purge THEN
			//Set the category Number
			IF Ldg[Bank].Found = 97 THEN // 97 is weight too small so always set to mixed so it doesn;t get sent to washer..
				myCat = CAT_MIXED_LINEN //Std.MaxCats	- 1
				myPrg = Std.MaxProg	- 1
			ELSE IF (myCat > 0) AND (Bag[StnBag].Cat <> myCat) THEN
				IF (MixCats OR MixProgs) THEN
					//Take the Cat code of bag with most weight
					IF (Bag[StnBag].Wgt > myWgt) THEN
						myCat = Bag[StnBag].Cat
						myPrg = Bag[StnBag].Prg
						myWgt = Bag[StnBag].Wgt
					ENDIF
				ELSE //Different Cats in 1 bag
					myCat = CAT_MIXED_LINEN//Std.MaxCats	- 1
					myPrg = Std.MaxProg - 1
				ENDIF
			ELSE
				myCat = Bag[StnBag].Cat
				myPrg = Bag[StnBag].Prg
				myWgt = Bag[StnBag].Wgt
			ENDIF

			IF (myCus > 0) AND (Bag[StnBag].Cus <> myCus) THEN
				myCus = Std.MaxCust - 1
			ELSE
				myCus = Bag[StnBag].Cus
			ENDIF
		ENDIF

		IF Purge AND (PurgeBagIndex = Std.PurgeBank[myBank].PurgeBagQty) THEN ;Do not minus 1 from purge qty as the indexing is above so will always read 1 more..
			Bag[myBag] 		= Bag[StnBag]
			Bag[StnBag].Mis = 0
			Bag[StnBag].Bid = 0 ; Reset BID

			Bag[myBag].Cat = myCat
			Bag[myBag].Prg = myPrg
			Bag[myBag].Ur2 = 99
			Bag[myBag].Cus	= myCus
			Bag[myBag].Dst 	= USINT(Ldg[myBank].Line)	;Destination
			Bag[myBag].Wgt 	= Std.PurgeBank[myBank].PurgeBatchWieght
			Bag[myBag].Cnt 	= Std.PurgeBank[myBank].PurgeBatchCount

			Bag[myBag].Timestamp = myTimeStamp
			Bag[StnBag].Bid = 0 ; Reset BID
			Bag[StnBag].Dst = 0 					;Reset Destination (Manual)
			Bag[StnBag].Mis = 0
			IF (Ldg[myBank].Found = 98) OR (Ldg[myBank].Found = 97) THEN
				D[900 + mySeq] = 3 ;Reverse belt not used.
			ELSE
				D[900 + mySeq] = 3
			ENDIF
		ELSE IF NOT Purge AND (Bag[StnBag].Cat <> 98) THEN
			;Copy Station Data to Belt Bag
			Bag[myBag] 		= Bag[StnBag]
			Bag[myBag].Dst 	= USINT(Ldg[myBank].Line)	;Destination
			Bag[myBag].Ur2 = StnBag
			Bag[StnBag].Bid = 0 ; Reset BID
			Bag[StnBag].Dst = 0 					;Reset Destination (Manual)
			Bag[StnBag].Mis = 0
			Bag[myBag].Timestamp = myTimeStamp
			D[900 + mySeq] = 3
		ENDIF
		Alarm[mySeq].Name = almNoAlarm
	ENDIF
ELSE
	Purge = FALSE
	PurgeBagIndex		= 0
	Ldg[myBank].Search  	= 0 ;Clear Search if not on step 2
	myCat = 0
	myPrg = 0
	myCus = 0
	myWgt = 0
ENDIF
ExitStep2:

;Get batch ID from SQL Server
IF ((STEP >= 3) AND (STEP <= 4)) THEN
	IF (Bag[myBag].Mis = 0) THEN
		_httpRequest;
	ENDIF
ELSE
	HTTP_Comm[myHttp].Status = HTTP_COMM_STATUS_DISABLED
ENDIF

;Step 3
;Release to Belt Conveyor
TON_10ms(I_PhotoTop,10,LinenDetected,LinenDetectedET)
IF (STEP = 3) THEN
	O_RunBelt = TRUE
	IF LinenDetected OR Test.TransferBelt THEN
		D[900 + mySeq] = 4
	ENDIF
	Alarm[mySeq].Name = almPhotocellNotMade
ENDIF

TON_10ms((STEP = 4),10,RunBelt,Step6ET)
IF (STEP = 4) THEN

	RequestRel.TransferBelt[myBelt] = (Bag[myBag].Cat > 0)
	n = D[900 + Std.StationBankReg + myBank]
	IF EnableRel.TransferBelt[myBelt] AND (ReportLoading[n].Cat = 0) THEN; AND (Bag[myBag].Mis > 0)
		;myTimeStamp = CurrentTimestamp
		ReportLoading[n].Prg = Bag[StnBag].Prg 			;Program
		ReportLoading[n].Cat = Bag[StnBag].Cat			;Category
		ReportLoading[n].Cus = Bag[StnBag].Cus			;Customer
		ReportLoading[n].Wgt = UINT(WeightValue)		;Weight
		ReportLoading[n].Cnt = UINT(CountValue)			;Count
		ReportLoading[n].Stn = n         				;Station
		ReportLoading[n].Mcn = 0						;Machine
		ReportLoading[n].Bid = Bag[StnBag].Bid			;Batch ID
		ReportLoading[n].Mis = Bag[myBag].Mis
		ReportLoading[n].TimeStamp = Bag[myBag].Timestamp
		D[900 + mySeq] = 5
	ENDIF
	IF (Bag[myBag].Cat = 0) THEN
		Alarm[mySeq].Name = almBagDataError
	ELSE IF (Bag[myBag].Mis = 0) THEN
		Alarm[mySeq].Name = almBagDataError
	ENDIF

ENDIF

;Step 5 - Run Belt until linen detected for 1 second and Station has emptied
TON_10ms(((STEP = 5) AND I_PhotoTop AND I_InvStatus),50,LinenIsDetected,LinenIsDetectedET)
IF (STEP = 5) THEN
	O_RunBelt = TRUE
	Ldg[myBank].EnableStnRelease = TRUE ;Enable Station to Open bags if they haven't been already
	IF (LinenIsDetected OR Test.TransferBelt)   THEN
		D[900 + mySeq] = 6
	ENDIF
	IF (Bag[myBag].Cat = 0) OR (Bag[myOutBag].Cat > 0) THEN
		Alarm[mySeq].Name = almBagDataError
	ELSE IF NOT Std.HaltSysZone[myZone] THEN
		Alarm[mySeq].Name = almPhotocellNotMade
	ENDIF
ENDIF

;Step 6 - Run Belt until photocells clear for 12 seconds
;TON_10ms((STEP = 6),200,MinimumRun,MinimumRunET)
TON_10ms(((STEP = 6) AND I_InvStatus  AND NOT I_PhotoTop AND NOT Std.HaltSysZone[myZone])AND MinBeltRun,1400,BeltClear,BeltClearET)
IF (STEP = 6) THEN
	O_RunBelt = TRUE
	IF (BeltClear AND (Bag[myBag].Cat > 0) AND ((Bag[myOutBag].Cat = 0) OR (Bag[myOutBag].Cat = Std.MaxCats))) THEN
		myBagNumber = Bag[myOutBag].Ur1
		Bag[myOutBag] = Bag[myBag]
		Bag[myOutBag].Ur1 = myBagNumber
		Bag[myBag] = Bag[0]
		D[900 + mySeq] = 7
	ENDIF
	IF NOT Std.HaltSysZone[myZone] THEN
		IF I_PhotoBottom OR I_PhotoTop THEN
			Alarm[mySeq].Name = almPhotocellBlocked
		ELSE IF StationOpen THEN
			Alarm[mySeq].Name = almStationNotClosed
		ELSE IF NOT MinBeltRun THEN
			Alarm[mySeq].Name = almClearingBeltPleaseWait
		ENDIF
	ENDIF
ENDIF

;Step  - Check Stations Are Closed
IF (STEP = 7) THEN
	IF NOT StationOpen AND (Bag[myBag].Cat = 0) THEN
		D[900 + mySeq] = 1
	ENDIF
	Alarm[mySeq].Name = almStationNotClosed
ENDIF

;Note - Unitl the Station has closed the min belt run time won't start
BeltRunTime = (7 + BeltAddTime)
;CTU((O_RunBelt AND Std.Clock1s AND (D[900 + Std.StationBankReg + myBank] = 0) AND NOT Std.EStop),(STEP = 1),BeltRunTime,MinBeltRun,MinBeltRunCV)
BeltRunning = (O_RunBelt OR O_Reverse)
CTU((BeltRunning AND I_InvStatus AND Std.Clock1s AND NOT StationOpen  AND NOT Std.HaltSysZone[myZone]),(STEP = 1),BeltRunTime,MinBeltRun,MinBeltRunCV)

;Slow speed for large load on belt
TON_10ms((NOT I_PhotoLarge AND NOT RunSlow),300,LargeLoadClear,LargeLoadClearET)
IF ((STEP > 2) AND (STEP < 7)) THEN
	IF I_PhotoLarge THEN
		O_SlowBelt = TRUE
	ENDIF
ENDIF

IF (STEP > 0) AND NOT I_InvStatus	THEN
	Alarm[mySeq].Name = almMotorOverload
	Alarm[mySeq].Time = 0
ENDIF

;Alarms
TimerAlarm.IN = NOT PLS AND (Alarm[mySeq].Name > 0)
TimerAlarm.PT = Alarm[mySeq].Time
TimerAlarm FUB TON_10ms()
Alarm[mySeq].On = TimerAlarm.Q
Alarm[mySeq].ET = TimerAlarm.ET

;Outputs
;Inform Station Sequences that the belt has been
Ldg[myBank].BeltHasRun =  (((((D[900 + mySeq] > 4) AND (D[900 + mySeq] < 7)) OR (D[900 + mySeq] >= 10)) AND Ldg[myBank].EnableStnRelease)  OR (D[900 + mySeq] = 1))

Y[365].Y02 = O_RunBelt
//Y[8].Y03 = O_RunBelt AND (STEP < 7) ; Inclined belt... Do not run when reversing.
//Y[8].Y02 = O_Reverse

END_PROGRAM
```

#### _httpRequest.st
```iecst
ACTION _httpRequest:
	myHttp := 6;

	CASE HTTP_Comm[myHttp].Status OF
		HTTP_COMM_STATUS_DISABLED:
			//Build Request String..
			itoa(Bag[myBag].Cat,ADR(catString));
			itoa(Bag[myBag].Cus,ADR(cusString));
			itoa(Bag[myBag].Wgt,ADR(wgtString));
			itoa(Bag[myBag].Mis,ADR(batchString));
			requestURL := HTTP_IF_CALL_USP_REPLY_URL;

			requestURL := CONCAT(requestURL,HTTP_GET_BATCH_CREATE);
			requestURL := CONCAT(requestURL,'@SystemIndex=');
			requestURL := CONCAT(requestURL,Std.PLCStnString);
			requestURL := CONCAT(requestURL,',@LocationIndex=0');
			requestURL := CONCAT(requestURL,',@CatID=');
			requestURL := CONCAT(requestURL,catString);
			requestURL := CONCAT(requestURL,',@CusID=');
			requestURL := CONCAT(requestURL,cusString);
			requestURL := CONCAT(requestURL,',@Wgt=');
			requestURL := CONCAT(requestURL,wgtString);

			HTTP_Comm[myHttp].Command.Method := httpMETHOD_GET;
			HTTP_Comm[myHttp].Command.Cmd_URL := requestURL;
			HTTP_Comm[myHttp].Command.Body_Data.Adr := 0;//ADR(requestData);
			HTTP_Comm[myHttp].Command.Body_Data.Size := 0;//SIZEOF(requestData);
			HTTP_Comm[myHttp].Command.ResponseData.Adr := ADR(responseData); ;
			HTTP_Comm[myHttp].Command.ResponseData.Size := SIZEOF(responseData);;
			HTTP_Comm[myHttp].Status := HTTP_COMM_STATUS_ACTIVE_WAIT_BUF;

		HTTP_COMM_STATUS_ACTIVE_WAIT_BUF:
			//Command is sent to ring buffer.
		HTTP_COMM_STATUS_IN_BUFFER:
			//Command recieved and in ring buffer
		HTTP_COMM_STATUS_IN_PROCESS:
			//Command being processed by httpClient.
		HTTP_COMM_STATUS_COMPLETE:
			//Decode response Data.
			//Response comes as Batch ID int, BatchID Guid.
			//Search for , that splits values
			commaPos := 0;
			FOR n := 1 TO 30 DO
				IF (responseData[n] = 44) THEN
					commaPos := n;
					EXIT;
				END_IF;
			END_FOR;
			IF (commaPos > 0) AND (commaPos <= 10) THEN // Check batch ID is in range.
				batchString := '';
				memcpy(ADR(batchString),ADR(responseData[1]),(commaPos -1 ));
				Bag[myBag].Mis := atoi(ADR(batchString));
			ELSE
				//Error with Batch ID or Proc has reutrn error...
				Alarm[mySeq].Name := ALM_BAG_DATA_ERROR;
				Alarm[mySeq].Time := 0;
			END_IF;

		//HTTP_Comm[myHttp].Status := HTTP_COMM_STATUS_DISABLED;

		HTTP_COMM_STATUS_ERROR:
			HTTP_Comm[myHttp].Status := HTTP_COMM_STATUS_DISABLED;

	END_CASE;

END_ACTION
```

#### _setBeltTime.st
```iecst
ACTION _setBeltTime:

BeltAddTimeArray[1] := 4;
BeltAddTimeArray[2] := 4;
BeltAddTimeArray[3] := 4;
BeltAddTimeArray[4] := 4;
BeltAddTimeArray[5] := 3;
BeltAddTimeArray[6] := 3;
BeltAddTimeArray[7] := 3;
BeltAddTimeArray[8] := 3;
BeltAddTimeArray[9] := 2;
BeltAddTimeArray[10] := 2;
BeltAddTimeArray[11] := 2;
BeltAddTimeArray[12] := 2;
BeltAddTimeArray[13] := 1;
BeltAddTimeArray[14] := 1;
BeltAddTimeArray[15] := 1;
BeltAddTimeArray[16] := 1;
BeltAddTimeArray[17] := 0;
BeltAddTimeArray[18] := 0;
BeltAddTimeArray[19] := 0;
BeltAddTimeArray[20] := 0;
BeltAddTimeArray[42] := 5;

END_ACTION
```

### constants.var - Local variables
```iecst
VAR CONSTANT
	MAX_ROTASTATIONS : USINT := 5;
END_VAR
VAR
	TON_SettledInStation : ARRAY[0..MAX_ROTASTATIONS] OF TON_10ms;
END_VAR
```

### Program Logical/BaseStandards/RotaSort/19_RotaSortContro (IEC) - *Empty base sequence

#### empty.var
```iecst
(********************************************************************
 * COPYRIGHT --
 ********************************************************************
 * Program: pr
 * File: pr.var
 * Author: treamsbottom
 * Created: July 16, 2015
 ********************************************************************
 * Local variables of program pr
 ********************************************************************)
VAR
	mySeq : UINT;
	myIO : UINT;
	myZone : UINT;
	myRelLine : UINT;
	myBag : UINT;
	i_bagAtBuffer : BOOL;
	i_bagAtBufferOut : BOOL;
	i_bufferOutOpen : BOOL;
	o_openBuffer : BOOL;
	step : UINT;
	pls : BOOL;
	timerAlarm : TON_10ms;
END_VAR
VAR RETAIN
	lastStep : UINT;
END_VAR
VAR
	bufferSettleTime : UDINT;
	myOutBag : UINT;
	myBank : UINT;
	ton_Reset : TON_10ms;
	lineValid : ARRAY[0..MAX_ROTASTATIONS] OF BOOL;
	waitTime : ARRAY[0..MAX_ROTASTATIONS] OF UDINT;
	waitingLongest : ARRAY[0..2] OF UDINT;
	o_reset : BOOL;
	ton_SettledBuffer : TON_10ms;
	bufferClear : BOOL;
	myStn : UINT;
	o_openStops : ARRAY[0..MAX_ROTASTATIONS] OF BOOL;
	i_bagOnStnA : ARRAY[0..MAX_ROTASTATIONS] OF BOOL;
	i_bagOnStnB : ARRAY[0..MAX_ROTASTATIONS] OF BOOL;
	o_Rotate : ARRAY[0..MAX_ROTASTATIONS] OF BOOL;
	StnBag : UINT;
	ton_Rotate : TON_10ms;
	o_openStopsRelease : ARRAY[0..MAX_ROTASTATIONS] OF BOOL;
	i_pastStop : ARRAY[0..MAX_ROTASTATIONS] OF BOOL;
	switchCheck : BOOL;
	closeStop : ARRAY[0..MAX_ROTASTATIONS] OF BOOL;
	bagAtBufferOut : BOOL;
	bufferOutOpen : BOOL;
	ton_FullBagTest : TON_10ms;
	ton_FullBagTest2 : TON_10ms;
	n : UINT;
	myStnBag : UINT;
	myBuffBag : UINT;
	recieveValid : BOOL;
	myInTransitBag : UINT;
	queueTime : ARRAY[0..2] OF UDINT;
	queueValid : ARRAY[0..2] OF BOOL;
END_VAR
```

#### empty.st
```iecst
(********************************************************************
 * COPYRIGHT --
 ********************************************************************
 * Program: pr
 * File: pr.st
 * Author: treamsbottom
 * Created: July 16, 2015
 ********************************************************************
 * Implementation of program pr
 ********************************************************************)
//V1.00.1 First Release
PROGRAM _INIT
//Configuration
mySeq						:= 19;	//Sequence number
myIO						:= 300; // Start of IO block for sorting stations - 1..
myZone						:= 1;
myBank						:= 1;
myBag						:= 219; //transit Bag
myBuffBag					:= 253;//Track empty bag in
myInTransitBag				:= 249;//Transit position for empty in ( Do not use if not tracking empty)
bufferSettleTime			:= 300;
myStnBag					:= 210; //Start or station bags (- 1) - The bags used when full, not the loading program)

myRelLine					:= 0;
myOutBag 					:= 221; //Line[myRelLine].LastBag;//Line[myRelLine].LastBag;
END_PROGRAM

PROGRAM _CYCLIC
//Inputs
i_bagAtBuffer				:= X[212].X03;

// Any Single bag buffer out IO.
bagAtBufferOut				:= X[32].X06;
bufferOutOpen				:= Y[32].Y08;

RequestRel.VC[1] := FALSE;

FOR n := 1 TO MAX_ROTASTATIONS  DO
	i_bagOnStnA[n]				:= X[myIO + n].X01;
	i_bagOnStnB[n]				:= X[myIO + n].X02;
	i_pastStop[n]				:= X[myIO + n].X04;
	o_openStops[n]				:= FALSE;
	o_openStopsRelease[n]		:= FALSE;
	o_Rotate[n]					:= FALSE;
	closeStop[n]				:= FALSE;
END_FOR;

o_openBuffer			:= FALSE;
o_reset					:= FALSE;

Ldg[myBank].EnableStnRelease := FALSE;

IF (myBag = 0) THEN
	Alarm[mySeq].Bag	:= mySeq + 10000;
ELSE
	Alarm[mySeq].Bag	:= myBag;
END_IF;

Alarm[mySeq].Name 		:= 0;
Alarm[mySeq].Beacon	:= TRUE;
Alarm[mySeq].Extra		:= 0;
Alarm[mySeq].Time		:= 3000;

//Global timers. Used in station for pusher type,
FOR n := 0 TO MAX_ROTASTATIONS DO
	TON_SettledInStation[n].IN := i_bagOnStnA[n] AND i_bagOnStnB[n];
	TON_SettledInStation[n].PT := 50;
	TON_SettledInStation[n]();
END_FOR;

//Setup Sequence
step := D[900 + mySeq];
//Setup Pulse contact
pls := (step <> lastStep);
lastStep := step;

//Sequence
IF (step = 0) THEN
	//Disabled
END_IF;

//Reset Points
ton_Reset.IN := (step = 1);
ton_Reset.PT := 150;
ton_Reset();
IF (step = 1) THEN
	D[950 + myBank]:= 0;
	o_reset := 1;
	switchCheck := 1;
	IF ton_Reset.Q THEN
		FOR n:= 1 TO MAX_ROTASTATIONS DO
			IF i_bagOnStnA[n] OR i_bagOnStnB[n] OR i_pastStop[n] THEN
				switchCheck := 0;
				EXIT;
			END_IF;
		END_FOR;
		IF switchCheck THEN
			Count[mySeq] := Count[mySeq] + 1;
			D[900 + mySeq] := 2;
		ELSE
			Alarm[mySeq].Name := ALM_SWITCH_FAULT;
		END_IF;
	END_IF;
END_IF;

//Waiting longest loop for sending empty into station
ton_SettledBuffer.IN := i_bagAtBuffer;
ton_SettledBuffer.PT := bufferSettleTime;
ton_SettledBuffer();
FOR n := Ldg[myBank].StartStn TO Ldg[myBank].EndStn DO
	lineValid[n] := Stn[n].requestBag;
	IF lineValid[n] THEN
		IF (waitTime[n] < 16#FFFFFFFF) THEN
			waitTime[n]:= waitTime[n] + 1;
		END_IF;
	ELSE
		waitTime[n] := 0;
	END_IF;
END_FOR;

waitingLongest[0] := 0;
waitTime[0] := 0;
FOR n := Ldg[myBank].StartStn TO Ldg[myBank].EndStn DO
	IF waitTime[n] > waitTime[0] THEN
		waitTime[0] := waitTime[n];
		waitingLongest[0] := n;
	END_IF;
END_FOR;

waitingLongest[1] := 0;
Stn[0].QTime := 0;
FOR n := Ldg[myBank].StartStn TO Ldg[myBank].EndStn DO
	IF Stn[n].QTime > Stn[0].QTime AND (Stn[n].QTime > 5) THEN // Settle 1 secs before releasing
		Stn[0].QTime := Stn[n].QTime;
		waitingLongest[1] := n;
	END_IF;
END_FOR;

//add next loop to decide which is waiting longest... Release bag or send bag.
FOR n:= 0 TO 1 DO
	IF waitingLongest[n] > 0 THEN
		IF (queueTime[n + 1] < 16#FFFFFFFF) THEN
			queueTime[n + 1]:= queueTime[n + 1] + 1;
		END_IF;
	ELSE
		queueTime[n + 1] := 0;
	END_IF;
END_FOR;
//..
bufferClear := Request.VC[1]; // Line[myRelLine].Clear AND (Bag[myOutBag].Cat = 0) AND NOT bufferOutOpen AND NOT bagAtBufferOut;
//step 2 = Decide what to do...
IF (step = 2) THEN
	IF (myBuffBag > 0) THEN
		recieveValid := ton_SettledBuffer.Q AND (Bag[myBuffBag].Cat > 0) AND (Bag[myInTransitBag].Cat = 0);
		IF (Bag[myInTransitBag].Cat > 0) THEN
			Alarm[mySeq].Name := ALM_BAG_DATA_ERROR;
			Alarm[mySeq].Bag := myInTransitBag;
			Alarm[mySeq].Time := 0;
		ELSIF ton_SettledBuffer.Q AND (Bag[myBuffBag].Cat = 0) THEN
			Alarm[mySeq].Name := ALM_BAG_DATA_ERROR;
			Alarm[mySeq].Bag := myBuffBag;
			Alarm[mySeq].Time := 500;
		END_IF;
	ELSE
		recieveValid := ton_SettledBuffer.Q;
	END_IF
	IF NOT Std.HaltSysZone[myZone] THEN
		//Decide if the Send or take bag based on wait time..
		queueValid[1] := recieveValid;
		queueValid[2] := bufferClear;
		waitingLongest[2] := 0;
		queueTime[0] := 0;
		FOR n := 1 TO 2 DO
			IF (queueTime[n] > queueTime[0]) AND queueValid[n] THEN
				queueTime[0] := queueTime[n];
				waitingLongest[2] := n;
			END_IF;
		END_FOR;
		//
		IF (waitingLongest[2] = 1) THEN//AND recieveValid THEN //Send empty bag
			D[950 + myBank] := UDINT_TO_UINT(waitingLongest[0]);
			IF (Bag[myBuffBag].Cat > 0) THEN
				Bag[myInTransitBag] := Bag[myBuffBag];
				Bag[myBuffBag] := Bag[0];
			END_IF;
			D[900 + mySeq] := 3;
		ELSIF (waitingLongest[2] = 2) THEN//AND bufferClear THEN	// Send Bag to Station
			D[950 + myBank] := UDINT_TO_UINT(waitingLongest[1]);
			D[900 + mySeq] := 7;
		END_IF;
	END_IF;
END_IF;

myStn := D[950 + myBank];
StnBag := myStnBag + myStn;
//step 3 select point to send
IF (step = 3) THEN
	o_openBuffer := TRUE;
	FOR n := 1 TO myStn DO // Open all stops down stream of stn.
		o_openStops[n] := TRUE;
	END_FOR;
	IF i_pastStop[myStn] THEN
		D[900 + mySeq] := 4;
	END_IF;
	Alarm[mySeq].Bag := myInTransitBag;
	Alarm[mySeq].Name := ALM_BAG_NOT_RELEASED;
    Alarm[mySeq].Time := 6000;
END_IF;

IF (step = 4) THEN
	closeStop[myStn] := 1;
	FOR n := 1 TO myStn DO // Open all stops down stream of stn.
		o_openStops[n] := TRUE;
	END_FOR;
	IF TON_SettledInStation[myStn].Q THEN
		D[900 + mySeq] := 5;
	END_IF;
	Alarm[mySeq].Bag := StnBag;
	Alarm[mySeq].Name := ALM_BAG_NOT_SETTLED;
    Alarm[mySeq].Time := 6000;
END_IF;

ton_Rotate.IN := (step = 5) OR (step = 7) OR (step = 9);
ton_Rotate.PT := 450;
ton_Rotate();
IF (step = 5) THEN
	o_Rotate[myStn] := TRUE;
	IF ton_Rotate.Q THEN
		D[900 + mySeq] := 6;
	END_IF;
END_IF;

IF (step = 6) THEN
	o_Rotate[myStn] := TRUE;
	o_openStops[myStn] := TRUE;
	IF NOT Stn[myStn].requestBag THEN
		IF (myBuffBag > 0) THEN
			Bag[StnBag] := Bag[myInTransitBag];
			Bag[myInTransitBag] := Bag[0];
		END_IF;
		D[900 + mySeq] := 1;
	END_IF;
	Alarm[mySeq].Name := ALM_BAG_NOT_RELEASED;
	Alarm[mySeq].Bag := StnBag;
    Alarm[mySeq].Time := 6000;
END_IF;

//Release Bag /Rotate Points..
IF (step = 7) THEN
	o_Rotate[myStn] := TRUE;
	IF ton_Rotate.Q THEN
		D[900 + mySeq] := 8;
	END_IF;

END_IF;

IF (step = 8) THEN
	Ldg[myBank].EnableStnRelease := TRUE;
	o_Rotate[myStn] := TRUE;
	IF 	(TON_SettledInStation[myStn].Q AND (Bag[myBag].Cat = 0) AND Stn[myStn].Unlock) AND Request.VC[1] THEN // Remove unlock if not using pusher type.
		IF (ReportLoading[myStn].Cat = 0) THEN
			Bag[myBag] := Bag[StnBag];
			Bag[StnBag] := Bag[0];
			ReportLoading[myStn].Prg := Bag[myBag].Prg;
			ReportLoading[myStn].Cat := Bag[myBag].Cat;
			ReportLoading[myStn].Cus := Bag[myBag].Cus;
			ReportLoading[myStn].Wgt := Bag[myBag].Wgt;
			ReportLoading[myStn].Cnt := 0;
			ReportLoading[myStn].Stn := myStn;
			ReportLoading[myStn].Mcn := 0;
			ReportLoading[myStn].Bid := Bag[myBag].Mis;
			D[900 + mySeq] := 9;
		END_IF;
		//C[myRelLine] := 0;
		//D[900 + mySeq] := 9;
	END_IF;
	Alarm[mySeq].Bag := StnBag;
	IF Bag[myBag].Cat > 0 THEN
		Alarm[mySeq].Name := ALM_BAG_DATA_ERROR;
	ELSIF NOT TON_SettledInStation[myStn].Q THEN
		Alarm[mySeq].Name := ALM_BAG_NOT_SETTLED;
        Alarm[mySeq].Time := 6000;
	END_IF;
END_IF;

//Release Bag /Rotate Points..
IF (step = 9) THEN
	IF ton_Rotate.Q THEN
		D[900 + mySeq] := 10;
	END_IF;
END_IF;

//Open Stations	bag arrives.
IF (step = 10) THEN
	FOR n := myStn TO MAX_ROTASTATIONS DO //Open all stop ahead of releasing station
		o_openStopsRelease[n] := TRUE;
	END_FOR;
	IF NOT Request.VC[1] AND (Bag[myBag].Cat = 0) THEN
		D[900 + mySeq] := 1;
	END_IF;
	Alarm[mySeq].Bag := myBag;
	Alarm[mySeq].Name := ALM_BAG_NOT_RELEASED;
    Alarm[mySeq].Time := 6000;
END_IF;

//-----------------------------------
//PLC Outputs - adjust TO suit system
//-----------------------------------

Y[212].Y06 := o_openBuffer;
FOR n := 1 TO MAX_ROTASTATIONS DO
	Y[myIO + n].Y07	:= o_Rotate[n];
	Y[myIO + n].Y08	:= ((o_openStops[n] OR o_openStopsRelease[n]) AND NOT closeStop[n]);
END_FOR;

//Alarms
timerAlarm(IN := NOT pls AND (Alarm[mySeq].Name > 0),PT:= Alarm[mySeq].Time);

Alarm[mySeq].On 	:= timerAlarm.Q;
Alarm[mySeq].ET 	:= timerAlarm.ET;

END_PROGRAM
```

### Program Logical/BaseStandards/RotaSort/RotaSortStn (IEC, version 1.00.1) - *Empty base sequence

#### empty.st - Implementation code
```iecst
(********************************************************************
 * COPYRIGHT --
 ********************************************************************
 * Program: pr
 * File: pr.st
 * Author: treamsbottom
 * Created: July 16, 2015
 ********************************************************************
 * Implementation of program pr
 ********************************************************************)
//V1.00.1 First Release
PROGRAM _INIT
myBank 						:= 1;
myZone						:= 1;
END_PROGRAM

PROGRAM _CYCLIC

i_partLoad[1]		:= X[306].X01;
i_partLoad[2]		:= X[306].X02;
i_partLoad[3]		:= X[306].X03;
i_partLoad[4]		:= X[306].X04;
i_partLoad[5]		:= X[307].X01;

FOR n := Ldg[myBank].StartStn  TO Ldg[myBank].EndStn DO
	//Configuration
	mySeq						:= 40;	//Sequence number
	myIO 						:= 300 + n;// Start of IO. will be auto incremented in control loop
	myBag						:= 210 + n;  //Start or station bags (- 1) - The bags used when full, not the loading program)
	//Keep in array size
	IF n > MAX_ROTASTATIONS THEN
		EXIT;
	END_IF;
	//Configuration
	myAlm					:= mySeq + n;// Alarm index
	mySeq					:= 900 + mySeq + n;	//Sequence number

	o_steady[n]			:= 0;
	o_releaseBag[n]		:= 0;
	o_pusher[n] 		:= 0;
	Stn[n].LampOn			:= 0;

	i_bagInStation[n] 	:= X[myIO].X03;

	Stn[n].requestBag	:= 0;
	Stn[n].Unlock 		:= 0;
	step := D[mySeq];
	ton_SettledStation[n].IN := (step = 4);//i_bagInStation[n];
	ton_SettledStation[n].PT := 150;
	ton_SettledStation[n]();

	StnBag := (Std.StationBagsStart[myBank] - 1  + n);

	IF (Bag[StnBag].Cat > 0) AND (Bag[StnBag].Bid = 0) AND (BidStn > 0) THEN
		Bag[StnBag].Bid := BidStn;
		BidStn := 0;
	END_IF;

	Bag[StnBag].Wgt := Stn[n].Weight;

	IF (StnBag = 0) THEN
		Alarm[myAlm].Bag	:= mySeq + 10000;
	ELSE
		Alarm[myAlm].Bag	:= StnBag;
	END_IF;

	Alarm[myAlm].Name 		:= 0;
	Alarm[myAlm].Beacon	    := TRUE;
	Alarm[myAlm].Extra		:= 0;
	Alarm[myAlm].Time		:= 3000;

	//Setup Sequence
	step := D[mySeq];
	//Setup Pulse contact
	pls := (step <> lastStep);
	lastStep := step;

	//Sequence
	IF (step = 0) THEN
		//Disabled
		Stn[n].QTime := 0;
		Stn[n].ManualRelease := 0;
		Stn[n].Purge := 0;
	END_IF;

	//1- Check station is empty
	IF (step = 1) THEN
		IF NOT 	i_bagInStation[n] AND (Bag[StnBag].Cat > 0) AND (Bag[myBag].Cat = 0) THEN// Make sure we have bag data from the loading prg..
			Stn[n].ManualRelease := 0;
			Stn[n].Purge := 0;
			Count[myAlm] := Count[myAlm] + 1;
			D[mySeq] := 2;
		ELSIF (Bag[myBag].Cat > 0) THEN
			Alarm[myAlm].Name := ALM_BAG_DATA_ERROR;
			Alarm[myAlm].Time := 6000;
			Alarm[myAlm].Bag := myBag;
		END_IF;
	END_IF;

	//2- Request Empty Bag
	IF (step = 2) THEN
		Stn[n].requestBag := TRUE;
		IF (D[950 + myBank] = n) THEN
			D[mySeq] := 3;
		END_IF;
	END_IF;

	//3- Bag enroute
	IF (step = 3) THEN
		Stn[n].requestBag := TRUE;
//		//Special for testing full bags only
//		o_pusher[n] := (D[950 + myBank] = n) AND Test_FullBagMode AND ((D[908] = 98) OR (D[908] = 99));
//		//End special
		IF i_bagInStation[n] THEN
			D[mySeq] := 4;
		END_IF;
		//Alarm Bag not arrived ?
	END_IF;

	//4 Bag arrives in station
	IF (step = 4) THEN
		IF ton_SettledStation[n].Q  AND (D[950 + myBank] <> n)  THEN
			D[mySeq] := 5;
		END_IF;
		Alarm[myAlm].Name := ALM_BAG_NOT_SETTLED;
	END_IF;

	o_steady[n] := (step > 4) AND (step <= 5) AND (Stn[n].Weight < 100);
	//5- Wieghing Step - Go in to Q
	IF (step = 5) THEN
		//When station goes into Q copy stn bag data into myBag
		IF i_partLoad[n] THEN
			Stn[n].ManualRelease := 1;
		END_IF;
		//Operate the lamp...(Red)
		Stn[n].LampOn := ((Stn[n].SP1 AND Std.Clock2s) OR Stn[n].SP2 OR (Stn[n].SP3 AND Std.Clock200ms));
		IF Stn[n].QTime > 30 AND ((Bag[myBag].Cat = 0) OR (Bag[myBag].Cat = Std.MaxCats)) AND (Bag[StnBag].Cat > 0) THEN
			myBagNumber := Bag[myBag].Ur2;
			Bag[myBag] := Bag[StnBag];
			Bag[myBag].Ur2 :=	myBagNumber;
			Bag[StnBag].Bid := 0;
		END_IF;
		IF (D[950 + myBank] = n) AND (Bag[myBag].Cat > 0) AND (Bag[myBag].Cat <> Std.MaxCats) AND Ldg[myBank].EnableStnRelease THEN
			D[mySeq] := 6;
		ELSIF (D[950 + myBank] = n) AND Ldg[myBank].EnableStnRelease THEN
			Alarm[myAlm].Name := ALM_BAG_DATA_ERROR;
            Alarm[myAlm].Time := 6000;
		END_IF;
	ELSE
		Stn[n].LampOn := 1;
	END_IF;

		ton_SettledWeight[n].IN := (step = 6);//i_bagInStation[n];
		ton_SettledWeight[n].PT := 150;
		ton_SettledWeight[n]();

	//6 Release Bag,,,
	IF (step = 6) THEN
	IF NOT ton_SettledWeight[n].Q THEN
		Bag[myBag].Wgt := Bag[StnBag].Wgt;
	END_IF;
	IF 	ton_SettledWeight[n].Q THEN
		o_releaseBag[n] := 1;
		IF TON_SettledInStation[n].Q THEN
			Bag[myBag].Timestamp := CurrentTimestamp;
			bagReleased[n] := 1;
		END_IF;
		o_pusher[n] := NOT bagReleased[n];
		Stn[n].Unlock := ton_retract[n].Q;
		IF (D[950 + myBank] <> n) THEN
			D[mySeq] := 1;
		END_IF;
	ELSE
			bagReleased[n] := 0;
	END_IF;
	END_IF;

//-----------------------------------
//PLC Outputs - adjust TO suit system
	//-----------------------------------
	//Remove if not using pusher...
	ton_retract[n].IN := NOT o_pusher[n];
	ton_retract[n].PT := 600;//
	ton_retract[n]();
	Y[myIO].Y05	:= o_reset;
	Y[myIO].Y06 := o_releaseBag[n];
	Y[myIO].Y05	:= o_pusher[n];

	//Alarms
	timerAlarm[n].IN := (Alarm[myAlm].Name > 0);
	timerAlarm[n].PT := Alarm[myAlm].Time;
	timerAlarm[n]();

	Alarm[myAlm].On 	:= timerAlarm[n].Q;
	Alarm[myAlm].ET 	:= timerAlarm[n].ET;

END_FOR;
Y[306].Y05 := Stn[1].LampOn;
Y[306].Y06 := Stn[2].LampOn;
Y[306].Y07 := Stn[3].LampOn;
Y[306].Y08 := Stn[4].LampOn;
Y[307].Y05 := Stn[5].LampOn;
Y[307].Y02 := o_steady[1];
Y[307].Y03 := o_steady[2];
Y[307].Y04 := o_steady[3];
Y[307].Y06 := o_steady[4];
Y[307].Y07 := o_steady[5];

END_PROGRAM
```

#### empty.var - Local variables
```iecst
(********************************************************************
 * COPYRIGHT --
 ********************************************************************
 * Program: pr
 * File: pr.var
 * Author: treamsbottom
 * Created: July 16, 2015
 ********************************************************************
 * Local variables of program pr
 ********************************************************************)
VAR
	mySeq : UINT;
	myIO : UINT;
	myZone : UINT;
	myRelLine : UINT;
	myBag : UINT;
	i_bagAtBuffer : BOOL;
	i_bagAtBufferOut : BOOL;
	i_bufferOutOpen : BOOL;
	o_openBuffer : BOOL;
	step : UINT;
	pls : BOOL;
	timerAlarm : ARRAY[0..MAX_ROTASTATIONS] OF TON_10ms;
END_VAR
VAR RETAIN
	lastStep : UINT;
END_VAR
VAR
	bufferSettleTime : UDINT;
	myOutBag : UINT;
	i_bagInStation : ARRAY[0..MAX_ROTASTATIONS] OF BOOL;
	myBank : UINT;
	ton_SettledStation : ARRAY[0..MAX_ROTASTATIONS] OF TON_10ms;
	o_steady : ARRAY[0..MAX_ROTASTATIONS] OF BOOL;
	o_releaseBag : ARRAY[0..MAX_ROTASTATIONS] OF BOOL;
	myAlm : UINT;
	ton_retract : ARRAY[0..MAX_ROTASTATIONS] OF TON_10ms;
	o_pusher : ARRAY[0..MAX_ROTASTATIONS] OF BOOL;
	bagReleased : ARRAY[0..MAX_ROTASTATIONS] OF BOOL;
	n : UINT;
	Test_FullBagMode : BOOL;
	StnBag : UINT;
	o_reset : BOOL;
	i_partLoad : ARRAY[0..MAX_ROTASTATIONS] OF BOOL;
	myBagNumber : UDINT;
	ton_SettledWeight : ARRAY[0..7] OF TON_10ms;
END_VAR
```

### Program Logical/BaseStandards/TwinRailLoadingUnit/lu_twin (IEC, version 1.01.1) - *Twin rail loading unit

#### lu.st - Implementation code
```iecst
(********************************************************************
 * COPYRIGHT --
 ********************************************************************
 * Program: lu twin rail loading unit
 * File: lu.st
 * Author: treamsbottom
 * Created: August 21, 2018
 ********************************************************************
 * Implementation of program lu
 ********************************************************************)
//V1.00.1 First Release
PROGRAM _INIT
//Configuration
mySeq						:= 30;	//Sequence number
myIO						:= 23;	//First IO Block
myLU						:= 2;	// Loading unit number
myZone						:= 1;	// Safety Zone
myBag						:= 201; //Buffer Bag
myBuffBag					:= 0; 	// Tracking Empty bag in...
myOutBag					:= 0; // there is a buffer after the loading unit.
useRequest					:= FALSE; //Use the Request bit. Only use when working with x_1_point. otherwise use RequestRelease as the i_bagAtBuffer.
bufferSettleTime			:= 300; // Time for bag to settle in buffer

useCompressor				:= FALSE;
myReportStn					:= 0;//myLU// Set Station index for reports. 0 = no report write.

myBelt						:= 1;	// Set if loaded by a belt
myCan						:= 0;	// Set if using Kanlink...

alarm						ACCESS ADR(Alarm[mySeq]);
bag							ACCESS ADR(Bag[myBag]);
bag_buff					ACCESS ADR(Bag[myBuffBag]);
bag_out						ACCESS ADR(Bag[myOutBag]);
can							ACCESS ADR(CAN[myCan]);

END_PROGRAM

PROGRAM _CYCLIC
//Inputs

i_bagInLoadingUnit[1]	:= X[myIO].X03;
i_bagInLoadingUnit[2]	:= X[myIO].X04;
i_bagAtBuffer[1]		:= X[myIO].X01;
i_bagAtBuffer[2]		:= X[myIO].X02;

i_compressorAtTop[1]	:= TRUE; // Set to TRUE if there is no compressor
i_compressorAtTop[2]	:= TRUE;
i_compress				:= FALSE;

i_bagAtBufferOut[1] 	:= FALSE;	// Is there a buffer after the loading unit..
i_bagAtBufferOut[2] 	:= FALSE;
i_bufferOutOpen[1]		:= FALSE;
i_bufferOutOpen[2]		:= FALSE;

o_openBuffer			:= FALSE;
o_steadyCylinders		:= FALSE;
o_releaseBag	 		:= FALSE;
o_moveCompressorDown	:= FALSE;

Request.LU[myLU]		:= FALSE;
RequestRel.LU[myLU]		:= FALSE;

IF (myBelt > 0) THEN
	EnableRel.TransferBelt[myBelt] := FALSE;
END_IF;

IF (myCan > 0) THEN
	can.ReadyToLoad := FALSE;
END_IF

IF (myBag = 0) THEN
	alarm.Bag	:= mySeq + 10000;
ELSE
	alarm.Bag	:= myBag;
END_IF;

alarm.Name 		:= 0;
alarm.Beacon		:= TRUE;
alarm.Extra		:= 0;
alarm.Time		:= 3000;

//Setup Sequence
step := D[900 + mySeq];
//Setup Pulse contact
pls := (step <> lastStep);
lastStep := step;

//Get BagID
IF (bag.Cat > 0) AND (bag.Bid = 0) AND (BidStn > 0) THEN
	bag.Bid := BidStn;
	BidStn := 0;
END_IF;

//Sequence
IF (step = 0) THEN
	//Disabled
END_IF;

lu_Enabled	:= (NOT Std.HaltSysZone[myZone]);//(D[mySeq] > 0) AND

//Check loading unit is clear.
switchFault 	:= (i_bagInLoadingUnit[1] OR i_bagInLoadingUnit[2]);
compressorUp 	:= (i_compressorAtTop[1] AND i_compressorAtTop[2]);
ton_10ms_LuClear(IN:= compressorUp AND NOT switchFault,PT:= 200);
IF (step = 1) THEN
	IF (ton_10ms_LuClear.Q AND lu_Enabled) THEN
		D[900 + mySeq] := 2;
		Count[mySeq] := Count[mySeq] + 1;
	END_IF;
	IF (switchFault OR NOT compressorUp) THEN
		alarm.Name := ALM_SWITCH_FAULT;
	END_IF;
END_IF;

// Step 2 - Wait for bag at buffer if used
ton_10ms_SettledBuffer(IN:= (i_bagAtBuffer[1] AND i_bagAtBuffer[2]), PT:= bufferSettleTime);
IF (step = 2) THEN
	IF useRequest THEN
		D[900 + mySeq] := 3;
	ELSE
		IF ton_10ms_SettledBuffer.Q THEN
			IF (myBuffBag > 0) THEN
				IF (bag_buff.Cat > 0) AND (bag.Cat = 0) THEN
					D[900 + mySeq] := 3;
				ELSIF (bag_buff.Cat = 0) THEN
					alarm.Name := ALM_BAG_DATA_ERROR;
					alarm.Bag := myBuffBag;
				ELSE
					alarm.Name := ALM_BAG_DATA_ERROR;
				END_IF;
			ELSE
				D[900 + mySeq] := 3;
			END_IF;
		ELSIF (myBuffBag > 0) AND (bag_buff.Cat > 0) THEN
			alarm.Name := ALM_BAG_NOT_SETTLED;
		END_IF;
	END_IF;
END_IF;

//Open buffer stop / Request bag
IF (step = 3) THEN
	releaseValid := ((myBuffBag = 0) OR ((bag.Cat = 0) AND (bag_buff.Cat > 0)));
	o_openBuffer := releaseValid AND NOT useRequest;
	Request.LU[myLU]  := releaseValid AND useRequest;
	IF ((i_bagInLoadingUnit[1] OR i_bagInLoadingUnit[2]) AND releaseValid) THEN
		IF (myBuffBag > 0) THEN
			bag := bag_buff; //Clear empty buffer bag data if used
			bag_buff := Bag[0];
		END_IF;
		D[900 + mySeq] := 4;
	ELSIF (myBuffBag > 0) THEN
		IF (bag.Cat > 0) THEN
			alarm.Name := ALM_BAG_DATA_ERROR;
			alarm.Time := 0;
		ELSIF (bag_buff.Cat = 0) THEN
			alarm.Name := ALM_BAG_DATA_ERROR;
			alarm.Bag := myBuffBag;
			alarm.Time := 0;
		ELSE
			alarm.Name  := ALM_BAG_NOT_ARRIVED;
		END_IF;
	ELSE
		alarm.Name  := ALM_BAG_NOT_ARRIVED;
	END_IF;
END_IF;

//Step 4 - Bag settles in loading unit
ton_10ms_SettleInLU(IN:= i_bagInLoadingUnit[1] AND i_bagInLoadingUnit[2] ,PT:= 300);
IF (step = 4) THEN
	IF ton_10ms_SettleInLU.Q THEN
		D[900 + mySeq] := 5;
	END_IF;
	alarm.Name := ALM_BAG_NOT_SETTLED;
END_IF;

//Steady cylinders on from steps 5 - 8
o_steadyCylinders := ((step >= 5) AND (step <= 8));

//Move Steady Cylinders down and check bag data
ton_10ms_SteadyDown(IN:= (step = 5), PT:= 200);
IF (step = 5) THEN
	IF ton_10ms_SteadyDown.Q  THEN
		IF (myBuffBag = 0) THEN
			IF (bag.Cat = 0) THEN
				D[900 + mySeq] := 6;
			ELSE
				alarm.Name := ALM_BAG_DATA_ERROR;
				alarm.Time := 0;
			END_IF;
		ELSE
			IF (bag.Cat = Std.MaxCats) THEN
				D[900 + mySeq] := 6;
			ELSE
				alarm.Name := ALM_BAG_DATA_ERROR;
				alarm.Time := 0;
			END_IF;
		END_IF;
	END_IF;
END_IF;

//Step 6 Wait for bag to be loaded..
IF (step = 6) THEN
	EnableRel.TransferBelt[myBelt] 	:= (myBelt > 0);
	IF (myCan > 0) THEN// Kanlink interface.
		can.ReadyToLoad 		:= NOT unloadFinished;
		IF (can.Category > 0) AND NOT unloadFinished THEN
			myPrg := UINT_TO_USINT(can.Program);
			myCat := can.Category;
			myCus := can.Customer;
			myWgt := can.Weight;
			myMis := can.BatchID;
		END_IF;
		// Get Program code
		IF ((myPrg = 0) AND (myCat > 0) AND (D32[100 + 20 * (myLU - 1)] <> myCat)) THEN
			D32[100 + 20 * (myLU - 1)] := myCat;
		ELSIF (D32[101 + 20 * (myLU - 1)] = myCat) THEN
			myPrg := UDINT_TO_USINT(D32[102 + 20 * (myLU - 1)]);
		END_IF;
		IF can.UnloadFinished THEN
			unloadFinished := TRUE;
		END_IF;
		IF (unloadFinished AND (myCat > 0) AND (myPrg > 0)) THEN
			bag.Prg := myPrg;
			bag.Cat := myCat;
			bag.Cus := myCus;
			bag.Wgt := myWgt;
			bag.Mis := myMis;
		END_IF;
	END_IF;

	IF (bag.Cat > 0) AND (bag.Prg > 0) AND ((bag.Cat <> Std.MaxCats) OR (myBuffBag = 0)) THEN
		IF (myReportStn > 0) THEN
			IF (ReportLoading[myReportStn].Cat = 0) THEN
				ReportLoading[myReportStn].Prg := bag.Prg;
				ReportLoading[myReportStn].Cat := bag.Cat;
				ReportLoading[myReportStn].Cus := bag.Cus;
				ReportLoading[myReportStn].Wgt := bag.Wgt;
				ReportLoading[myReportStn].Cnt := 0;
				ReportLoading[myReportStn].Stn := myReportStn;
				ReportLoading[myReportStn].Mcn := 0;
				ReportLoading[myReportStn].Bid := bag.Mis;
				D[900 + mySeq] := 7;
			END_IF;
		ELSE
			D[900 + mySeq] := 7;
		END_IF;
	ELSIF (myCan > 0) AND unloadFinished THEN
		alarm.Name := ALM_BAG_DATA_ERROR;
	END_IF;
ELSE
	D32[100 + 20 * (myLU - 1)] := 0;
	unloadFinished := FALSE;
	can.ReadyToLoad := FALSE;
	can.Program := 0;
	can.Category := 0;
	can.Customer := 0;
	can.Weight := 0;
	can.BatchID := 0;
END_IF;

//Step 7 Check If compression is required
ton_10ms_CompressCheck(IN:=(step = 7),PT:= 30);
IF (step = 7) THEN
	IF useCompressor THEN
		IF i_compress THEN
			compress := TRUE;
		END_IF;
		IF ton_10ms_CompressCheck.Q THEN
			IF compress THEN
				D[900 + mySeq] := 8; // Compress
			ELSE
				D[900 + mySeq] := 9;	// Check compressor is OK
			END_IF;
		END_IF;
	ELSE
		D[900 + mySeq] := 9;
	END_IF;
ELSE
	compress := FALSE;
END_IF;

//Step 8 move linen compressor down.
ton_10ms_CompressDown(IN:=(step = 8),PT:= 500);
IF (step = 8) THEN
	IF useCompressor THEN
		IF ton_10ms_CompressDown.Q THEN
			D[900 + mySeq] := 9;
		END_IF;
	ELSE
		D[900 + mySeq] := 9;
	END_IF;
END_IF;

//step 9 check compressor status
ton_10ms_CompressorCheck(IN:=((i_compressorAtTop[1] AND i_compressorAtTop[2]) OR NOT useCompressor),PT:= 200);
IF (step = 9) THEN
	IF ton_10ms_CompressorCheck.Q  AND NOT Std.HaltSysZone[myZone] THEN
		D[900 + mySeq] := 10;
	END_IF;
	alarm.Name := ALM_SWITCH_FAULT;
END_IF;

//Check for line space.
IF (step = 10) THEN
	releaseValid := (NOT i_bagAtBufferOut[1] AND NOT i_bufferOutOpen[1] AND NOT i_bagAtBufferOut[2] AND NOT i_bufferOutOpen[2] AND (bag.Cat > 0) AND (bag_out.Cat = 0));
	IF NOT Std.HaltSysZone[myZone] THEN
		IF (myOutBag > 0) THEN // We are releasing into a buffer after the loading unit.
			IF releaseValid THEN
				D[900 + mySeq] := 11;
			END_IF;
		ELSE
			RequestRel.LU[myLU] := releaseValid;
			IF EnableRel.LU[myLU] AND releaseValid THEN
				D[900 + mySeq] := 11;
			END_IF;
		END_IF;
		IF (myBag > 0) AND (bag.Cat = 0) THEN
			alarm.Name := ALM_BAG_DATA_ERROR;
			alarm.Time := 0;
		END_IF;
	END_IF;
END_IF;

//Release bag.
IF (step = 11) THEN

	IF (myOutBag > 0) THEN
		releaseValid := (NOT i_bagAtBufferOut[1] AND NOT i_bufferOutOpen[1] AND NOT i_bagAtBufferOut[2] AND NOT i_bufferOutOpen[2] AND (bag.Cat > 0) AND (bag_out.Cat = 0));
		o_releaseBag := releaseValid;
		IF i_bagAtBufferOut[1] AND i_bagAtBufferOut[2] THEN
			IF (bag.Cat > 0) AND (bag_out.Cat = 0) THEN
				bag_out := bag;
				bag := Bag[0];
				D[900 + mySeq] := 1;
			ELSE
				alarm.Name := ALM_BAG_DATA_ERROR;
				alarm.Time := 0;
			END_IF;
		ELSIF releaseValid THEN
			alarm.Name := ALM_BAG_NOT_RELEASED;
		END_IF;
	ELSE // We are using request and enable..
		o_releaseBag := EnableRel.LU[myLU];
		IF NOT EnableRel.LU[myLU] AND (bag.Cat = 0) THEN // Make sure data is copied out by enabling sequence.
			D[900 + mySeq] := 1;
		ELSIF NOT EnableRel.LU[myLU] AND (bag.Cat > 0) THEN
			alarm.Name := ALM_BAG_DATA_ERROR;
		END_IF;
	END_IF;
END_IF;

//-----------------------------------
//PLC Outputs - adjust TO suit system
//-----------------------------------

Y[myIO].Y07 		:= o_releaseBag;
Y[myIO].Y08 		:= o_releaseBag;

Y[myIO].Y05 		:= o_openBuffer;
Y[myIO].Y06 		:= o_openBuffer;

Y[myIO + 1].Y05 	:= o_steadyCylinders;
Y[myIO + 1].Y06 	:= o_steadyCylinders; //Elephants foot

//Y[myIO + 1].Y07 	:= o_moveCompressorDown;
//Y[myIO + 1].Y08 	:= o_moveCompressorDown;

//Alarms
timerAlarm(IN := NOT pls AND (alarm.Name > 0),PT:= alarm.Time);

alarm.On 	:= timerAlarm.Q;
alarm.ET 	:= timerAlarm.ET;

END_PROGRAM
```

#### lu.var - Local variables
```iecst
(********************************************************************
 * COPYRIGHT --
 ********************************************************************
 * Program: lu
 * File: lu.var
 * Author: treamsbottom
 * Created: July 17, 2015
 ********************************************************************
 * Local variables of program lu
 ********************************************************************)
VAR
	useRequest : BOOL;
	useCompressor : BOOL;
	ton_10ms_SteadyDown : TON_10ms;
	ton_10ms_SettleInLU : TON_10ms;
	timerAlarm : TON_10ms;
	switchFault : BOOL;
	step : UINT;
	releaseValid : BOOL;
	pls : BOOL;
	o_steadyCylinders : BOOL;
	o_openBuffer : BOOL;
	o_moveCompressorDown : BOOL;
	myZone : UINT;
	mySeq : UINT;
	myOutBag : UINT;
	myLU : UINT;
	myIO : UINT;
	myBuffBag : UINT;
	myBag : UINT;
	lu_Enabled : BOOL;
END_VAR
VAR RETAIN
	lastStep : UINT;
END_VAR
VAR
	i_compressorAtTop : ARRAY[0..2] OF BOOL;
	i_compress : BOOL;
	i_bufferOutOpen : ARRAY[0..2] OF BOOL;
	i_bagInLoadingUnit : ARRAY[0..2] OF BOOL;
	i_bagAtBufferOut : ARRAY[0..2] OF BOOL;
	i_bagAtBuffer : ARRAY[0..2] OF BOOL;
	compressorUp : BOOL;
	compress : BOOL;
	bufferSettleTime : UINT;
	myReportStn : UINT;
	myBelt : UINT;
	myCan : UINT;
	unloadFinished : BOOL;
	ton_10ms_LuClear : TON_10ms;
	ton_10ms_SettledBuffer : TON_10ms;
	ton_10ms_CompressCheck : TON_10ms;
	ton_10ms_CompressDown : TON_10ms;
	ton_10ms_CompressorCheck : TON_10ms;
	myPrg : USINT;
	myCat : UDINT;
	myCus : UDINT;
	myWgt : UINT;
	myMis : UDINT;
	alarm : REFERENCE TO Alm;
	bag : REFERENCE TO Bag_typ;
	bag_out : REFERENCE TO Bag_typ;
	bag_buff : REFERENCE TO Bag_typ;
	can : REFERENCE TO CAN_Vars;
	o_releaseBag : BOOL := 0;
END_VAR
```

### Program Logical/BaseStandards/TwinRailLoadingUnit/lpn (IEC, version 1.00.1) - *Twin rail loading ongoing
